(* Logix 5000 project; controller reports 1756-L63 rev 20.15; software revision 20.04; part 34 of 52 *)

        [22].log_data[35].max := 1.0, [22].log_data[35].total := 1322.998, [22].log_data[35].time := 3600.0, [22].log_data[35].minminute := 3, [22].log_data[35].valid := 1, [22].log_data[36].max := 1.0, [22].log_data[36].total := 1539.2471, [22].log_data[36].time := 3600.0, [22].log_data[36].maxminute := 5, [22].log_data[36].valid := 1, [22].log_data[37].time := 3600.0, [22].log_data[37].valid := 1, [22].log_data[38].time := 3600.0, [22].log_data[38].valid := 1, [22].log_data[39].min := 0.9938818, [22].log_data[39].max := 1.0064838, [22].log_data[39].total := 3605.8333, [22].log_data[39].time := 3600.0, [22].log_data[39].minminute := 45, [22].log_data[39].maxminute := 14, [22].log_data[39].valid := 1, [22].log_data[40].min := 7.5643167, [22].log_data[40].max := 7.586301, [22].log_data[40].total := 27282.406, [22].log_data[40].time := 3600.0, [22].log_data[40].minminute := 14, [22].log_data[40].maxminute := 26, [22].log_data[40].valid := 1, [22].log_data[41].min := 0.032943603, [22].log_data[41].max := 0.058854003, [22].log_data[41].total := 164.49648, [22].log_data[41].time := 3600.0, [22].log_data[41].minminute := 22, [22].log_data[41].valid := 1, [22].log_data[42].min := 2.291996, [22].log_data[42].max := 2.297767, [22].log_data[42].total := 8263.503, [22].log_data[42].time := 3600.0, [22].log_data[42].minminute := 32, [22].log_data[42].maxminute := 12, [22].log_data[42].valid := 1, [22].log_data[43].min := -0.26000214, [22].log_data[43].max := -0.26000214, [22].log_data[43].total := -935.9732, [22].log_data[43].time := 3600.0, [22].log_data[43].valid := 1, [22].log_data[44].min := -0.30000305, [22].log_data[44].max := -0.27999878, [22].log_data[44].total := -1015.7973, [22].log_data[44].time := 3600.0, [22].log_data[44].valid := 1, [22].log_data[45].time := 3600.0, [22].log_data[45].valid := 1, [22].log_data[46].time := 3600.0, [22].log_data[46].valid := 1, [22].log_data[47].time := 3600.0, [22].log_data[47].valid := 1, [22].log_data[48].min := 6.7563815, [22].log_data[48].max := 6.7984266, [22].log_data[48].total := 24360.947,
        [22].log_data[48].time := 3600.0, [22].log_data[48].minminute := 57, [22].log_data[48].valid := 1, [22].log_data[49].min := 8.905314, [22].log_data[49].max := 9.548168, [22].log_data[49].total := 33928.742, [22].log_data[49].time := 3600.0, [22].log_data[49].maxminute := 53, [22].log_data[49].valid := 1, [22].log_data[50].min := 1.9997966, [22].log_data[50].max := 2.0873032, [22].log_data[50].total := 7348.6255, [22].log_data[50].time := 3600.0, [22].log_data[50].minminute := 54, [22].log_data[50].maxminute := 59, [22].log_data[50].valid := 1, [22].log_data[51].time := 3600.0, [22].log_data[51].valid := 1, [22].log_data[52].min := -2.7799988, [22].log_data[52].max := 0.13999939, [22].log_data[52].total := -7224.4995, [22].log_data[52].time := 3600.0, [22].log_data[52].minminute := 27, [22].log_data[52].valid := 1, [22].log_data[53].min := -2.7000046, [22].log_data[53].max := 0.19999695, [22].log_data[53].total := -6896.3794, [22].log_data[53].time := 3600.0, [22].log_data[53].minminute := 16, [22].log_data[53].maxminute := 5, [22].log_data[53].valid := 1, [22].log_data[54].max := 0.537, [22].log_data[54].total := 1118.8905, [22].log_data[54].time := 3600.0, [22].log_data[54].valid := 1, [22].log_data[55].max := 0.5575, [22].log_data[55].total := 1135.9928, [22].log_data[55].time := 3600.0, [22].log_data[55].minminute := 3, [22].log_data[55].maxminute := 16, [22].log_data[55].valid := 1, [22].log_data[56].min := 0.16024561, [22].log_data[56].max := 0.1607167, [22].log_data[56].total := 577.52075, [22].log_data[56].time := 3600.0, [22].log_data[56].minminute := 12, [22].log_data[56].maxminute := 46, [22].log_data[56].valid := 1, [22].log_data[57].min := 0.3022821, [22].log_data[57].max := 0.30271393, [22].log_data[57].total := 1088.9108, [22].log_data[57].time := 3600.0, [22].log_data[57].minminute := 44, [22].log_data[57].maxminute := 4, [22].log_data[57].valid := 1, [22].log_data[58].time := 3600.0, [22].log_data[58].valid := 1, [22].log_data[59].time := 3600.0, [22].log_data[59].valid := 1, [22].log_data[60].valid := 1,
        [22].log_data[61].valid := 1, [22].log_data[62].valid := 1, [22].log_data[63].valid := 1, [22].log_data[64].valid := 1, [22].log_data[65].valid := 1, [22].log_data[66].valid := 1, [22].log_data[67].valid := 1, [22].log_data[68].valid := 1, [22].log_data[69].valid := 1, [22].log_data[70].valid := 1, [22].log_data[71].valid := 1, [22].log_data[72].valid := 1, [22].log_data[73].valid := 1, [22].log_data[74].valid := 1, [22].log_data[75].valid := 1, [22].log_data[76].valid := 1, [22].log_data[77].valid := 1, [22].log_data[78].valid := 1, [22].log_data[79].valid := 1, [22].log_data[80].valid := 1, [22].log_data[81].valid := 1, [22].log_data[82].valid := 1, [22].log_data[83].valid := 1, [22].log_data[84].valid := 1, [22].log_data[85].valid := 1, [22].log_data[86].valid := 1, [22].log_data[87].valid := 1, [22].log_data[88].valid := 1, [22].log_data[89].valid := 1, [22].log_data[90].valid := 1, [22].log_data[91].valid := 1, [22].log_data[92].valid := 1, [22].log_data[93].valid := 1, [22].log_data[94].valid := 1, [22].log_data[95].valid := 1, [22].log_data[96].valid := 1, [22].log_data[97].valid := 1, [22].log_data[98].valid := 1, [22].log_data[99].valid := 1, [22].log_data[100].valid := 1, [22].log_data[101].valid := 1, [22].log_data[102].valid := 1, [22].log_data[103].valid := 1, [22].log_data[104].valid := 1, [22].log_data[105].valid := 1, [22].log_data[106].valid := 1, [22].log_data[107].valid := 1, [22].log_data[108].valid := 1, [22].log_data[109].valid := 1, [22].log_data[110].valid := 1, [22].log_data[111].valid := 1, [22].log_data[112].valid := 1, [22].log_data[113].valid := 1, [22].log_data[114].valid := 1, [22].log_data[115].valid := 1, [22].log_data[116].valid := 1, [22].log_data[117].valid := 1, [22].log_data[118].valid := 1, [22].log_data[119].valid := 1, [22].log_data[120].valid := 1,
        [22].log_data[121].valid := 1, [22].log_data[122].valid := 1, [22].log_data[123].valid := 1, [22].log_data[124].valid := 1, [22].time.Year := 2023, [22].time.Month := 1, [22].time.Day := 14, [22].time.Hour := 1, [22].time.Minute := 59, [22].time.Second := 59, [23].log_data[0].min := 1.0, [23].log_data[0].max := 1.0, [23].log_data[0].total := 3600.0, [23].log_data[0].time := 3600.0, [23].log_data[0].valid := 1, [23].log_data[1].max := 1.0, [23].log_data[1].total := 523.5, [23].log_data[1].time := 3600.0, [23].log_data[1].maxminute := 36, [23].log_data[1].valid := 1, [23].log_data[2].max := 1.0, [23].log_data[2].total := 520.0, [23].log_data[2].time := 3600.0, [23].log_data[2].maxminute := 36, [23].log_data[2].valid := 1, [23].log_data[3].time := 3600.0, [23].log_data[3].valid := 1, [23].log_data[4].time := 3600.0, [23].log_data[4].valid := 1, [23].log_data[5].max := 1.0, [23].log_data[5].total := 229.5, [23].log_data[5].time := 3600.0, [23].log_data[5].maxminute := 39, [23].log_data[5].valid := 1, [23].log_data[6].time := 3600.0, [23].log_data[6].valid := 1, [23].log_data[7].time := 3600.0, [23].log_data[7].valid := 1, [23].log_data[8].max := 1.0, [23].log_data[8].total := 1148.249, [23].log_data[8].time := 3600.0, [23].log_data[8].maxminute := 40, [23].log_data[8].valid := 1, [23].log_data[9].max := 1.0, [23].log_data[9].total := 1144.749, [23].log_data[9].time := 3600.0, [23].log_data[9].maxminute := 40, [23].log_data[9].valid := 1, [23].log_data[10].min := 1.0, [23].log_data[10].max := 1.0, [23].log_data[10].total := 3600.0, [23].log_data[10].time := 3600.0, [23].log_data[10].valid := 1, [23].log_data[11].time := 3600.0, [23].log_data[11].valid := 1, [23].log_data[12].min := 1.0, [23].log_data[12].max := 1.0, [23].log_data[12].total := 3600.0, [23].log_data[12].time := 3600.0, [23].log_data[12].valid := 1,
        [23].log_data[13].min := 1.0, [23].log_data[13].max := 1.0, [23].log_data[13].total := 3600.0, [23].log_data[13].time := 3600.0, [23].log_data[13].valid := 1, [23].log_data[14].time := 3600.0, [23].log_data[14].valid := 1, [23].log_data[15].time := 3600.0, [23].log_data[15].valid := 1, [23].log_data[16].time := 3600.0, [23].log_data[16].valid := 1, [23].log_data[17].min := 1.0, [23].log_data[17].max := 1.0, [23].log_data[17].total := 3600.0, [23].log_data[17].time := 3600.0, [23].log_data[17].valid := 1, [23].log_data[18].time := 3600.0, [23].log_data[18].valid := 1, [23].log_data[19].time := 3600.0, [23].log_data[19].valid := 1, [23].log_data[20].time := 3600.0, [23].log_data[20].valid := 1, [23].log_data[21].min := 1.0, [23].log_data[21].max := 1.0, [23].log_data[21].total := 3600.0, [23].log_data[21].time := 3600.0, [23].log_data[21].valid := 1, [23].log_data[22].time := 3600.0, [23].log_data[22].valid := 1, [23].log_data[23].time := 3600.0, [23].log_data[23].valid := 1, [23].log_data[24].time := 3600.0, [23].log_data[24].valid := 1, [23].log_data[25].time := 3600.0, [23].log_data[25].valid := 1, [23].log_data[26].time := 3600.0, [23].log_data[26].valid := 1, [23].log_data[27].time := 3600.0, [23].log_data[27].valid := 1, [23].log_data[28].time := 3600.0, [23].log_data[28].valid := 1, [23].log_data[29].min := 1.0, [23].log_data[29].max := 1.0, [23].log_data[29].total := 3600.0, [23].log_data[29].time := 3600.0, [23].log_data[29].valid := 1, [23].log_data[30].min := 1.0, [23].log_data[30].max := 1.0, [23].log_data[30].total := 3600.0, [23].log_data[30].time := 3600.0, [23].log_data[30].valid := 1, [23].log_data[31].max := 1.0, [23].log_data[31].total := 434.5, [23].log_data[31].time := 3600.0, [23].log_data[31].maxminute := 40, [23].log_data[31].valid := 1, [23].log_data[32].max := 1.0, [23].log_data[32].total := 543.249, [23].log_data[32].time := 3600.0, [23].log_data[32].maxminute := 49,
        [23].log_data[32].valid := 1, [23].log_data[33].time := 3600.0, [23].log_data[33].valid := 1, [23].log_data[34].time := 3600.0, [23].log_data[34].valid := 1, [23].log_data[35].max := 1.0, [23].log_data[35].total := 417.998, [23].log_data[35].time := 3600.0, [23].log_data[35].maxminute := 41, [23].log_data[35].valid := 1, [23].log_data[36].max := 1.0, [23].log_data[36].total := 543.249, [23].log_data[36].time := 3600.0, [23].log_data[36].maxminute := 44, [23].log_data[36].valid := 1, [23].log_data[37].max := 7.614469, [23].log_data[37].total := 3441.945, [23].log_data[37].time := 3600.0, [23].log_data[37].maxminute := 38, [23].log_data[37].valid := 1, [23].log_data[38].time := 3600.0, [23].log_data[38].valid := 1, [23].log_data[39].min := 0.9950596, [23].log_data[39].max := 1.02203, [23].log_data[39].total := 3610.5056, [23].log_data[39].time := 3600.0, [23].log_data[39].minminute := 11, [23].log_data[39].maxminute := 43, [23].log_data[39].valid := 1, [23].log_data[40].min := 7.5431566, [23].log_data[40].max := 7.5961943, [23].log_data[40].total := 27280.893, [23].log_data[40].time := 3600.0, [23].log_data[40].minminute := 4, [23].log_data[40].maxminute := 36, [23].log_data[40].valid := 1, [23].log_data[41].min := 0.030784423, [23].log_data[41].max := 0.052769043, [23].log_data[41].total := 143.54086, [23].log_data[41].time := 3600.0, [23].log_data[41].minminute := 33, [23].log_data[41].maxminute := 9, [23].log_data[41].valid := 1, [23].log_data[42].min := 2.291996, [23].log_data[42].max := 2.2975314, [23].log_data[42].total := 8263.341, [23].log_data[42].time := 3600.0, [23].log_data[42].minminute := 5, [23].log_data[42].maxminute := 10, [23].log_data[42].valid := 1, [23].log_data[43].min := -0.26000214, [23].log_data[43].max := -0.26000214, [23].log_data[43].total := -935.9732, [23].log_data[43].time := 3600.0, [23].log_data[43].valid := 1, [23].log_data[44].min := -0.30000305, [23].log_data[44].max := -0.27999878, [23].log_data[44].total := -1011.4277, [23].log_data[44].time := 3600.0, [23].log_data[44].valid := 1,
        [23].log_data[45].time := 3600.0, [23].log_data[45].valid := 1, [23].log_data[46].time := 3600.0, [23].log_data[46].valid := 1, [23].log_data[47].time := 3600.0, [23].log_data[47].valid := 1, [23].log_data[48].min := 6.665145, [23].log_data[48].max := 6.9523196, [23].log_data[48].total := 24385.578, [23].log_data[48].time := 3600.0, [23].log_data[48].minminute := 59, [23].log_data[48].maxminute := 45, [23].log_data[48].valid := 1, [23].log_data[49].min := 7.0688124, [23].log_data[49].max := 9.542084, [23].log_data[49].total := 32485.41, [23].log_data[49].time := 3600.0, [23].log_data[49].minminute := 59, [23].log_data[49].maxminute := 3, [23].log_data[49].valid := 1, [23].log_data[50].min := 2.0678706, [23].log_data[50].max := 2.1526685, [23].log_data[50].total := 7561.778, [23].log_data[50].time := 3600.0, [23].log_data[50].minminute := 43, [23].log_data[50].maxminute := 40, [23].log_data[50].valid := 1, [23].log_data[51].time := 3600.0, [23].log_data[51].valid := 1, [23].log_data[52].min := -4.1800003, [23].log_data[52].max := 0.11999512, [23].log_data[52].total := -6155.475, [23].log_data[52].time := 3600.0, [23].log_data[52].minminute := 41, [23].log_data[52].maxminute := 48, [23].log_data[52].valid := 1, [23].log_data[53].min := -3.9799957, [23].log_data[53].max := 0.19999695, [23].log_data[53].total := -5728.4756, [23].log_data[53].time := 3600.0, [23].log_data[53].minminute := 41, [23].log_data[53].maxminute := 54, [23].log_data[53].valid := 1, [23].log_data[54].max := 0.5275, [23].log_data[54].total := 387.55862, [23].log_data[54].time := 3600.0, [23].log_data[54].maxminute := 49, [23].log_data[54].valid := 1, [23].log_data[55].max := 0.5285, [23].log_data[55].total := 378.56726, [23].log_data[55].time := 3600.0, [23].log_data[55].maxminute := 54, [23].log_data[55].valid := 1, [23].log_data[56].min := 0.16024561, [23].log_data[56].max := 0.1607167, [23].log_data[56].total := 577.70746, [23].log_data[56].time := 3600.0, [23].log_data[56].minminute := 54, [23].log_data[56].maxminute := 30, [23].log_data[56].valid := 1,
        [23].log_data[57].min := 0.30232134, [23].log_data[57].max := 0.30275318, [23].log_data[57].total := 1088.9501, [23].log_data[57].time := 3600.0, [23].log_data[57].maxminute := 43, [23].log_data[57].valid := 1, [23].log_data[58].time := 3600.0, [23].log_data[58].valid := 1, [23].log_data[59].time := 3600.0, [23].log_data[59].valid := 1, [23].log_data[60].valid := 1, [23].log_data[61].valid := 1, [23].log_data[62].valid := 1, [23].log_data[63].valid := 1, [23].log_data[64].valid := 1, [23].log_data[65].valid := 1, [23].log_data[66].valid := 1, [23].log_data[67].valid := 1, [23].log_data[68].valid := 1, [23].log_data[69].valid := 1, [23].log_data[70].valid := 1, [23].log_data[71].valid := 1, [23].log_data[72].valid := 1, [23].log_data[73].valid := 1, [23].log_data[74].valid := 1, [23].log_data[75].valid := 1, [23].log_data[76].valid := 1, [23].log_data[77].valid := 1, [23].log_data[78].valid := 1, [23].log_data[79].valid := 1, [23].log_data[80].valid := 1, [23].log_data[81].valid := 1, [23].log_data[82].valid := 1, [23].log_data[83].valid := 1, [23].log_data[84].valid := 1, [23].log_data[85].valid := 1, [23].log_data[86].valid := 1, [23].log_data[87].valid := 1, [23].log_data[88].valid := 1, [23].log_data[89].valid := 1, [23].log_data[90].valid := 1, [23].log_data[91].valid := 1, [23].log_data[92].valid := 1, [23].log_data[93].valid := 1, [23].log_data[94].valid := 1, [23].log_data[95].valid := 1, [23].log_data[96].valid := 1, [23].log_data[97].valid := 1, [23].log_data[98].valid := 1, [23].log_data[99].valid := 1, [23].log_data[100].valid := 1, [23].log_data[101].valid := 1, [23].log_data[102].valid := 1, [23].log_data[103].valid := 1, [23].log_data[104].valid := 1, [23].log_data[105].valid := 1, [23].log_data[106].valid := 1, [23].log_data[107].valid := 1, [23].log_data[108].valid := 1, [23].log_data[109].valid := 1,
        [23].log_data[110].valid := 1, [23].log_data[111].valid := 1, [23].log_data[112].valid := 1, [23].log_data[113].valid := 1, [23].log_data[114].valid := 1, [23].log_data[115].valid := 1, [23].log_data[116].valid := 1, [23].log_data[117].valid := 1, [23].log_data[118].valid := 1, [23].log_data[119].valid := 1, [23].log_data[120].valid := 1, [23].log_data[121].valid := 1, [23].log_data[122].valid := 1, [23].log_data[123].valid := 1, [23].log_data[124].valid := 1, [23].time.Year := 2023, [23].time.Month := 1, [23].time.Day := 14, [23].time.Hour := 2, [23].time.Minute := 59, [23].time.Second := 59, [24].log_data[0].min := 1.0, [24].log_data[0].max := 1.0, [24].log_data[0].total := 3600.0, [24].log_data[0].time := 3600.0, [24].log_data[0].valid := 1, [24].log_data[1].time := 3600.0, [24].log_data[1].valid := 1, [24].log_data[2].time := 3600.0, [24].log_data[2].valid := 1, [24].log_data[3].time := 3600.0, [24].log_data[3].valid := 1, [24].log_data[4].time := 3600.0, [24].log_data[4].valid := 1, [24].log_data[5].time := 3600.0, [24].log_data[5].valid := 1, [24].log_data[6].time := 3600.0, [24].log_data[6].valid := 1, [24].log_data[7].time := 3600.0, [24].log_data[7].valid := 1, [24].log_data[8].min := 1.0, [24].log_data[8].max := 1.0, [24].log_data[8].total := 3600.0, [24].log_data[8].time := 3600.0, [24].log_data[8].valid := 1, [24].log_data[9].min := 1.0, [24].log_data[9].max := 1.0, [24].log_data[9].total := 3600.0, [24].log_data[9].time := 3600.0, [24].log_data[9].valid := 1, [24].log_data[10].min := 1.0, [24].log_data[10].max := 1.0, [24].log_data[10].total := 3600.0, [24].log_data[10].time := 3600.0, [24].log_data[10].valid := 1, [24].log_data[11].time := 3600.0, [24].log_data[11].valid := 1, [24].log_data[12].min := 1.0, [24].log_data[12].max := 1.0, [24].log_data[12].total := 3600.0,
        [24].log_data[12].time := 3600.0, [24].log_data[12].valid := 1, [24].log_data[13].min := 1.0, [24].log_data[13].max := 1.0, [24].log_data[13].total := 3600.0, [24].log_data[13].time := 3600.0, [24].log_data[13].valid := 1, [24].log_data[14].time := 3600.0, [24].log_data[14].valid := 1, [24].log_data[15].time := 3600.0, [24].log_data[15].valid := 1, [24].log_data[16].time := 3600.0, [24].log_data[16].valid := 1, [24].log_data[17].min := 1.0, [24].log_data[17].max := 1.0, [24].log_data[17].total := 3600.0, [24].log_data[17].time := 3600.0, [24].log_data[17].valid := 1, [24].log_data[18].time := 3600.0, [24].log_data[18].valid := 1, [24].log_data[19].time := 3600.0, [24].log_data[19].valid := 1, [24].log_data[20].time := 3600.0, [24].log_data[20].valid := 1, [24].log_data[21].min := 1.0, [24].log_data[21].max := 1.0, [24].log_data[21].total := 3600.0, [24].log_data[21].time := 3600.0, [24].log_data[21].valid := 1, [24].log_data[22].time := 3600.0, [24].log_data[22].valid := 1, [24].log_data[23].time := 3600.0, [24].log_data[23].valid := 1, [24].log_data[24].time := 3600.0, [24].log_data[24].valid := 1, [24].log_data[25].time := 3600.0, [24].log_data[25].valid := 1, [24].log_data[26].time := 3600.0, [24].log_data[26].valid := 1, [24].log_data[27].time := 3600.0, [24].log_data[27].valid := 1, [24].log_data[28].time := 3600.0, [24].log_data[28].valid := 1, [24].log_data[29].min := 1.0, [24].log_data[29].max := 1.0, [24].log_data[29].total := 3600.0, [24].log_data[29].time := 3600.0, [24].log_data[29].valid := 1, [24].log_data[30].min := 1.0, [24].log_data[30].max := 1.0, [24].log_data[30].total := 3600.0, [24].log_data[30].time := 3600.0, [24].log_data[30].valid := 1, [24].log_data[31].max := 1.0, [24].log_data[31].total := 1629.7471, [24].log_data[31].time := 3600.0, [24].log_data[31].valid := 1, [24].log_data[32].max := 1.0, [24].log_data[32].total := 1515.7471, [24].log_data[32].time := 3600.0,
        [24].log_data[32].maxminute := 10, [24].log_data[32].valid := 1, [24].log_data[33].time := 3600.0, [24].log_data[33].valid := 1, [24].log_data[34].time := 3600.0, [24].log_data[34].valid := 1, [24].log_data[35].max := 1.0, [24].log_data[35].total := 1440.7471, [24].log_data[35].time := 3600.0, [24].log_data[35].minminute := 3, [24].log_data[35].valid := 1, [24].log_data[36].max := 1.0, [24].log_data[36].total := 1629.7471, [24].log_data[36].time := 3600.0, [24].log_data[36].maxminute := 5, [24].log_data[36].valid := 1, [24].log_data[37].time := 3600.0, [24].log_data[37].valid := 1, [24].log_data[38].time := 3600.0, [24].log_data[38].valid := 1, [24].log_data[39].min := 0.9945885, [24].log_data[39].max := 1.0074259, [24].log_data[39].total := 3607.058, [24].log_data[39].time := 3600.0, [24].log_data[39].minminute := 14, [24].log_data[39].maxminute := 34, [24].log_data[39].valid := 1, [24].log_data[40].min := 7.5717363, [24].log_data[40].max := 7.586301, [24].log_data[40].total := 27285.361, [24].log_data[40].time := 3600.0, [24].log_data[40].minminute := 3, [24].log_data[40].maxminute := 5, [24].log_data[40].valid := 1, [24].log_data[41].min := 0.029017823, [24].log_data[41].max := 0.047469236, [24].log_data[41].total := 144.30215, [24].log_data[41].time := 3600.0, [24].log_data[41].minminute := 46, [24].log_data[41].maxminute := 11, [24].log_data[41].valid := 1, [24].log_data[42].min := 2.292585, [24].log_data[42].max := 2.297767, [24].log_data[42].total := 8263.188, [24].log_data[42].time := 3600.0, [24].log_data[42].minminute := 8, [24].log_data[42].maxminute := 13, [24].log_data[42].valid := 1, [24].log_data[43].min := -0.26000214, [24].log_data[43].max := -0.26000214, [24].log_data[43].total := -935.9732, [24].log_data[43].time := 3600.0, [24].log_data[43].valid := 1, [24].log_data[44].min := -0.30000305, [24].log_data[44].max := -0.27999878, [24].log_data[44].total := -1011.2831, [24].log_data[44].time := 3600.0, [24].log_data[44].valid := 1, [24].log_data[45].time := 3600.0, [24].log_data[45].valid := 1,
        [24].log_data[46].time := 3600.0, [24].log_data[46].valid := 1, [24].log_data[47].time := 3600.0, [24].log_data[47].valid := 1, [24].log_data[48].min := 6.595069, [24].log_data[48].max := 6.7967777, [24].log_data[48].total := 24212.92, [24].log_data[48].time := 3600.0, [24].log_data[48].minminute := 10, [24].log_data[48].maxminute := 25, [24].log_data[48].valid := 1, [24].log_data[49].min := 6.9688993, [24].log_data[49].max := 9.5318775, [24].log_data[49].total := 31036.44, [24].log_data[49].time := 3600.0, [24].log_data[49].minminute := 2, [24].log_data[49].maxminute := 58, [24].log_data[49].valid := 1, [24].log_data[50].min := 2.006863, [24].log_data[50].max := 2.0901299, [24].log_data[50].total := 7375.6206, [24].log_data[50].time := 3600.0, [24].log_data[50].minminute := 59, [24].log_data[50].valid := 1, [24].log_data[51].time := 3600.0, [24].log_data[51].valid := 1, [24].log_data[52].min := -3.040001, [24].log_data[52].max := 0.13999939, [24].log_data[52].total := -7732.567, [24].log_data[52].time := 3600.0, [24].log_data[52].minminute := 42, [24].log_data[52].maxminute := 40, [24].log_data[52].valid := 1, [24].log_data[53].min := -2.5, [24].log_data[53].max := 0.22000122, [24].log_data[53].total := -7008.48, [24].log_data[53].time := 3600.0, [24].log_data[53].minminute := 18, [24].log_data[53].maxminute := 4, [24].log_data[53].valid := 1, [24].log_data[54].max := 0.5645, [24].log_data[54].total := 1246.528, [24].log_data[54].time := 3600.0, [24].log_data[54].maxminute := 42, [24].log_data[54].valid := 1, [24].log_data[55].max := 0.538, [24].log_data[55].total := 1217.1504, [24].log_data[55].time := 3600.0, [24].log_data[55].minminute := 3, [24].log_data[55].maxminute := 47, [24].log_data[55].valid := 1, [24].log_data[56].min := 0.16024561, [24].log_data[56].max := 0.16079521, [24].log_data[56].total := 577.71893, [24].log_data[56].time := 3600.0, [24].log_data[56].minminute := 56, [24].log_data[56].maxminute := 32, [24].log_data[56].valid := 1, [24].log_data[57].min := 0.30079022, [24].log_data[57].max := 0.30271393,
        [24].log_data[57].total := 1084.8229, [24].log_data[57].time := 3600.0, [24].log_data[57].minminute := 47, [24].log_data[57].valid := 1, [24].log_data[58].time := 3600.0, [24].log_data[58].valid := 1, [24].log_data[59].time := 3600.0, [24].log_data[59].valid := 1, [24].log_data[60].valid := 1, [24].log_data[61].valid := 1, [24].log_data[62].valid := 1, [24].log_data[63].valid := 1, [24].log_data[64].valid := 1, [24].log_data[65].valid := 1, [24].log_data[66].valid := 1, [24].log_data[67].valid := 1, [24].log_data[68].valid := 1, [24].log_data[69].valid := 1, [24].log_data[70].valid := 1, [24].log_data[71].valid := 1, [24].log_data[72].valid := 1, [24].log_data[73].valid := 1, [24].log_data[74].valid := 1, [24].log_data[75].valid := 1, [24].log_data[76].valid := 1, [24].log_data[77].valid := 1, [24].log_data[78].valid := 1, [24].log_data[79].valid := 1, [24].log_data[80].valid := 1, [24].log_data[81].valid := 1, [24].log_data[82].valid := 1, [24].log_data[83].valid := 1, [24].log_data[84].valid := 1, [24].log_data[85].valid := 1, [24].log_data[86].valid := 1, [24].log_data[87].valid := 1, [24].log_data[88].valid := 1, [24].log_data[89].valid := 1, [24].log_data[90].valid := 1, [24].log_data[91].valid := 1, [24].log_data[92].valid := 1, [24].log_data[93].valid := 1, [24].log_data[94].valid := 1, [24].log_data[95].valid := 1, [24].log_data[96].valid := 1, [24].log_data[97].valid := 1, [24].log_data[98].valid := 1, [24].log_data[99].valid := 1, [24].log_data[100].valid := 1, [24].log_data[101].valid := 1, [24].log_data[102].valid := 1, [24].log_data[103].valid := 1, [24].log_data[104].valid := 1, [24].log_data[105].valid := 1, [24].log_data[106].valid := 1, [24].log_data[107].valid := 1, [24].log_data[108].valid := 1, [24].log_data[109].valid := 1, [24].log_data[110].valid := 1, [24].log_data[111].valid := 1,
        [24].log_data[112].valid := 1, [24].log_data[113].valid := 1, [24].log_data[114].valid := 1, [24].log_data[115].valid := 1, [24].log_data[116].valid := 1, [24].log_data[117].valid := 1, [24].log_data[118].valid := 1, [24].log_data[119].valid := 1, [24].log_data[120].valid := 1, [24].log_data[121].valid := 1, [24].log_data[122].valid := 1, [24].log_data[123].valid := 1, [24].log_data[124].valid := 1, [24].time.Year := 2023, [24].time.Month := 1, [24].time.Day := 14, [24].time.Hour := 3, [24].time.Minute := 59, [24].time.Second := 59, [25].log_data[0].min := 1.0, [25].log_data[0].max := 1.0, [25].log_data[0].total := 3600.0, [25].log_data[0].time := 3600.0, [25].log_data[0].valid := 1, [25].log_data[1].time := 3600.0, [25].log_data[1].valid := 1, [25].log_data[2].time := 3600.0, [25].log_data[2].valid := 1, [25].log_data[3].time := 3600.0, [25].log_data[3].valid := 1, [25].log_data[4].time := 3600.0, [25].log_data[4].valid := 1, [25].log_data[5].time := 3600.0, [25].log_data[5].valid := 1, [25].log_data[6].time := 3600.0, [25].log_data[6].valid := 1, [25].log_data[7].time := 3600.0, [25].log_data[7].valid := 1, [25].log_data[8].max := 1.0, [25].log_data[8].total := 227.751, [25].log_data[8].time := 3600.0, [25].log_data[8].minminute := 3, [25].log_data[8].valid := 1, [25].log_data[9].max := 1.0, [25].log_data[9].total := 227.751, [25].log_data[9].time := 3600.0, [25].log_data[9].minminute := 3, [25].log_data[9].valid := 1, [25].log_data[10].min := 1.0, [25].log_data[10].max := 1.0, [25].log_data[10].total := 3600.0, [25].log_data[10].time := 3600.0, [25].log_data[10].valid := 1, [25].log_data[11].time := 3600.0, [25].log_data[11].valid := 1, [25].log_data[12].min := 1.0, [25].log_data[12].max := 1.0, [25].log_data[12].total := 3600.0, [25].log_data[12].time := 3600.0, [25].log_data[12].valid := 1,
        [25].log_data[13].min := 1.0, [25].log_data[13].max := 1.0, [25].log_data[13].total := 3600.0, [25].log_data[13].time := 3600.0, [25].log_data[13].valid := 1, [25].log_data[14].time := 3600.0, [25].log_data[14].valid := 1, [25].log_data[15].time := 3600.0, [25].log_data[15].valid := 1, [25].log_data[16].time := 3600.0, [25].log_data[16].valid := 1, [25].log_data[17].min := 1.0, [25].log_data[17].max := 1.0, [25].log_data[17].total := 3600.0, [25].log_data[17].time := 3600.0, [25].log_data[17].valid := 1, [25].log_data[18].time := 3600.0, [25].log_data[18].valid := 1, [25].log_data[19].time := 3600.0, [25].log_data[19].valid := 1, [25].log_data[20].time := 3600.0, [25].log_data[20].valid := 1, [25].log_data[21].min := 1.0, [25].log_data[21].max := 1.0, [25].log_data[21].total := 3600.0, [25].log_data[21].time := 3600.0, [25].log_data[21].valid := 1, [25].log_data[22].time := 3600.0, [25].log_data[22].valid := 1, [25].log_data[23].time := 3600.0, [25].log_data[23].valid := 1, [25].log_data[24].time := 3600.0, [25].log_data[24].valid := 1, [25].log_data[25].time := 3600.0, [25].log_data[25].valid := 1, [25].log_data[26].time := 3600.0, [25].log_data[26].valid := 1, [25].log_data[27].time := 3600.0, [25].log_data[27].valid := 1, [25].log_data[28].time := 3600.0, [25].log_data[28].valid := 1, [25].log_data[29].min := 1.0, [25].log_data[29].max := 1.0, [25].log_data[29].total := 3600.0, [25].log_data[29].time := 3600.0, [25].log_data[29].valid := 1, [25].log_data[30].min := 1.0, [25].log_data[30].max := 1.0, [25].log_data[30].total := 3600.0, [25].log_data[30].time := 3600.0, [25].log_data[30].valid := 1, [25].log_data[31].max := 1.0, [25].log_data[31].total := 29.249, [25].log_data[31].time := 3600.0, [25].log_data[31].maxminute := 3, [25].log_data[31].valid := 1, [25].log_data[32].max := 1.0, [25].log_data[32].total := 114.0, [25].log_data[32].time := 3600.0, [25].log_data[32].minminute := 1,
        [25].log_data[32].valid := 1, [25].log_data[33].time := 3600.0, [25].log_data[33].valid := 1, [25].log_data[34].time := 3600.0, [25].log_data[34].valid := 1, [25].log_data[35].max := 1.0, [25].log_data[35].total := 231.5, [25].log_data[35].time := 3600.0, [25].log_data[35].minminute := 3, [25].log_data[35].valid := 1, [25].log_data[36].time := 3600.0, [25].log_data[36].valid := 1, [25].log_data[37].time := 3600.0, [25].log_data[37].valid := 1, [25].log_data[38].time := 3600.0, [25].log_data[38].valid := 1, [25].log_data[39].min := 0.9945885, [25].log_data[39].max := 1.0076615, [25].log_data[39].total := 3606.9658, [25].log_data[39].time := 3600.0, [25].log_data[39].minminute := 56, [25].log_data[39].maxminute := 27, [25].log_data[39].valid := 1, [25].log_data[40].min := 7.5643167, [25].log_data[40].max := 7.587675, [25].log_data[40].total := 27287.488, [25].log_data[40].time := 3600.0, [25].log_data[40].minminute := 47, [25].log_data[40].maxminute := 27, [25].log_data[40].valid := 1, [25].log_data[41].min := 0.034906495, [25].log_data[41].max := 0.05963916, [25].log_data[41].total := 160.86324, [25].log_data[41].time := 3600.0, [25].log_data[41].maxminute := 49, [25].log_data[41].valid := 1, [25].log_data[42].min := 2.2922316, [25].log_data[42].max := 2.2974136, [25].log_data[42].total := 8263.044, [25].log_data[42].time := 3600.0, [25].log_data[42].minminute := 25, [25].log_data[42].maxminute := 36, [25].log_data[42].valid := 1, [25].log_data[43].min := -0.26000214, [25].log_data[43].max := -0.26000214, [25].log_data[43].total := -935.9732, [25].log_data[43].time := 3600.0, [25].log_data[43].valid := 1, [25].log_data[44].min := -0.30000305, [25].log_data[44].max := -0.27999878, [25].log_data[44].total := -1009.182, [25].log_data[44].time := 3600.0, [25].log_data[44].valid := 1, [25].log_data[45].time := 3600.0, [25].log_data[45].valid := 1, [25].log_data[46].time := 3600.0, [25].log_data[46].valid := 1, [25].log_data[47].time := 3600.0, [25].log_data[47].valid := 1, [25].log_data[48].min := 6.7492356,
        [25].log_data[48].max := 6.762702, [25].log_data[48].total := 24321.047, [25].log_data[48].time := 3600.0, [25].log_data[48].minminute := 5, [25].log_data[48].maxminute := 52, [25].log_data[48].valid := 1, [25].log_data[49].min := 9.508125, [25].log_data[49].max := 9.581735, [25].log_data[49].total := 34331.49, [25].log_data[49].time := 3600.0, [25].log_data[49].minminute := 7, [25].log_data[49].maxminute := 57, [25].log_data[49].valid := 1, [25].log_data[50].min := 1.9999144, [25].log_data[50].max := 2.1099162, [25].log_data[50].total := 7540.0083, [25].log_data[50].time := 3600.0, [25].log_data[50].minminute := 3, [25].log_data[50].maxminute := 54, [25].log_data[50].valid := 1, [25].log_data[51].time := 3600.0, [25].log_data[51].valid := 1, [25].log_data[52].min := -2.7400055, [25].log_data[52].max := 0.11999512, [25].log_data[52].total := -5230.148, [25].log_data[52].time := 3600.0, [25].log_data[52].minminute := 3, [25].log_data[52].maxminute := 2, [25].log_data[52].valid := 1, [25].log_data[53].min := -2.4800034, [25].log_data[53].max := -0.16000366, [25].log_data[53].total := -5175.728, [25].log_data[53].time := 3600.0, [25].log_data[53].maxminute := 3, [25].log_data[53].valid := 1, [25].log_data[54].max := 0.505, [25].log_data[54].total := 55.965687, [25].log_data[54].time := 3600.0, [25].log_data[54].minminute := 1, [25].log_data[54].maxminute := 3, [25].log_data[54].valid := 1, [25].log_data[55].max := 0.44349998, [25].log_data[55].total := 93.022255, [25].log_data[55].time := 3600.0, [25].log_data[55].minminute := 3, [25].log_data[55].valid := 1, [25].log_data[56].min := 0.16028486, [25].log_data[56].max := 0.16079521, [25].log_data[56].total := 577.82935, [25].log_data[56].time := 3600.0, [25].log_data[56].minminute := 2, [25].log_data[56].maxminute := 7, [25].log_data[56].valid := 1, [25].log_data[57].min := 0.3008295, [25].log_data[57].max := 0.30126134, [25].log_data[57].total := 1083.6661, [25].log_data[57].time := 3600.0, [25].log_data[57].minminute := 3, [25].log_data[57].maxminute := 28, [25].log_data[57].valid := 1,
        [25].log_data[58].time := 3600.0, [25].log_data[58].valid := 1, [25].log_data[59].time := 3600.0, [25].log_data[59].valid := 1, [25].log_data[60].valid := 1, [25].log_data[61].valid := 1, [25].log_data[62].valid := 1, [25].log_data[63].valid := 1, [25].log_data[64].valid := 1, [25].log_data[65].valid := 1, [25].log_data[66].valid := 1, [25].log_data[67].valid := 1, [25].log_data[68].valid := 1, [25].log_data[69].valid := 1, [25].log_data[70].valid := 1, [25].log_data[71].valid := 1, [25].log_data[72].valid := 1, [25].log_data[73].valid := 1, [25].log_data[74].valid := 1, [25].log_data[75].valid := 1, [25].log_data[76].valid := 1, [25].log_data[77].valid := 1, [25].log_data[78].valid := 1, [25].log_data[79].valid := 1, [25].log_data[80].valid := 1, [25].log_data[81].valid := 1, [25].log_data[82].valid := 1, [25].log_data[83].valid := 1, [25].log_data[84].valid := 1, [25].log_data[85].valid := 1, [25].log_data[86].valid := 1, [25].log_data[87].valid := 1, [25].log_data[88].valid := 1, [25].log_data[89].valid := 1, [25].log_data[90].valid := 1, [25].log_data[91].valid := 1, [25].log_data[92].valid := 1, [25].log_data[93].valid := 1, [25].log_data[94].valid := 1, [25].log_data[95].valid := 1, [25].log_data[96].valid := 1, [25].log_data[97].valid := 1, [25].log_data[98].valid := 1, [25].log_data[99].valid := 1, [25].log_data[100].valid := 1, [25].log_data[101].valid := 1, [25].log_data[102].valid := 1, [25].log_data[103].valid := 1, [25].log_data[104].valid := 1, [25].log_data[105].valid := 1, [25].log_data[106].valid := 1, [25].log_data[107].valid := 1, [25].log_data[108].valid := 1, [25].log_data[109].valid := 1, [25].log_data[110].valid := 1, [25].log_data[111].valid := 1, [25].log_data[112].valid := 1, [25].log_data[113].valid := 1, [25].log_data[114].valid := 1, [25].log_data[115].valid := 1,
        [25].log_data[116].valid := 1, [25].log_data[117].valid := 1, [25].log_data[118].valid := 1, [25].log_data[119].valid := 1, [25].log_data[120].valid := 1, [25].log_data[121].valid := 1, [25].log_data[122].valid := 1, [25].log_data[123].valid := 1, [25].log_data[124].valid := 1, [25].time.Year := 2023, [25].time.Month := 1, [25].time.Day := 14, [25].time.Hour := 4, [25].time.Minute := 59, [25].time.Second := 59, [26].log_data[0].min := 1.0, [26].log_data[0].max := 1.0, [26].log_data[0].total := 3600.0, [26].log_data[0].time := 3600.0, [26].log_data[0].valid := 1, [26].log_data[1].time := 3600.0, [26].log_data[1].valid := 1, [26].log_data[2].time := 3600.0, [26].log_data[2].valid := 1, [26].log_data[3].time := 3600.0, [26].log_data[3].valid := 1, [26].log_data[4].time := 3600.0, [26].log_data[4].valid := 1, [26].log_data[5].time := 3600.0, [26].log_data[5].valid := 1, [26].log_data[6].time := 3600.0, [26].log_data[6].valid := 1, [26].log_data[7].time := 3600.0, [26].log_data[7].valid := 1, [26].log_data[8].time := 3600.0, [26].log_data[8].valid := 1, [26].log_data[9].time := 3600.0, [26].log_data[9].valid := 1, [26].log_data[10].min := 1.0, [26].log_data[10].max := 1.0, [26].log_data[10].total := 3600.0, [26].log_data[10].time := 3600.0, [26].log_data[10].valid := 1, [26].log_data[11].time := 3600.0, [26].log_data[11].valid := 1, [26].log_data[12].min := 1.0, [26].log_data[12].max := 1.0, [26].log_data[12].total := 3600.0, [26].log_data[12].time := 3600.0, [26].log_data[12].valid := 1, [26].log_data[13].min := 1.0, [26].log_data[13].max := 1.0, [26].log_data[13].total := 3600.0, [26].log_data[13].time := 3600.0, [26].log_data[13].valid := 1, [26].log_data[14].time := 3600.0, [26].log_data[14].valid := 1, [26].log_data[15].time := 3600.0, [26].log_data[15].valid := 1, [26].log_data[16].time := 3600.0,
        [26].log_data[16].valid := 1, [26].log_data[17].min := 1.0, [26].log_data[17].max := 1.0, [26].log_data[17].total := 3600.0, [26].log_data[17].time := 3600.0, [26].log_data[17].valid := 1, [26].log_data[18].time := 3600.0, [26].log_data[18].valid := 1, [26].log_data[19].time := 3600.0, [26].log_data[19].valid := 1, [26].log_data[20].time := 3600.0, [26].log_data[20].valid := 1, [26].log_data[21].min := 1.0, [26].log_data[21].max := 1.0, [26].log_data[21].total := 3600.0, [26].log_data[21].time := 3600.0, [26].log_data[21].valid := 1, [26].log_data[22].time := 3600.0, [26].log_data[22].valid := 1, [26].log_data[23].time := 3600.0, [26].log_data[23].valid := 1, [26].log_data[24].time := 3600.0, [26].log_data[24].valid := 1, [26].log_data[25].time := 3600.0, [26].log_data[25].valid := 1, [26].log_data[26].time := 3600.0, [26].log_data[26].valid := 1, [26].log_data[27].time := 3600.0, [26].log_data[27].valid := 1, [26].log_data[28].time := 3600.0, [26].log_data[28].valid := 1, [26].log_data[29].min := 1.0, [26].log_data[29].max := 1.0, [26].log_data[29].total := 3600.0, [26].log_data[29].time := 3600.0, [26].log_data[29].valid := 1, [26].log_data[30].min := 1.0, [26].log_data[30].max := 1.0, [26].log_data[30].total := 3600.0, [26].log_data[30].time := 3600.0, [26].log_data[30].valid := 1, [26].log_data[31].time := 3600.0, [26].log_data[31].valid := 1, [26].log_data[32].time := 3600.0, [26].log_data[32].valid := 1, [26].log_data[33].time := 3600.0, [26].log_data[33].valid := 1, [26].log_data[34].time := 3600.0, [26].log_data[34].valid := 1, [26].log_data[35].time := 3600.0, [26].log_data[35].valid := 1, [26].log_data[36].time := 3600.0, [26].log_data[36].valid := 1, [26].log_data[37].time := 3600.0, [26].log_data[37].valid := 1, [26].log_data[38].time := 3600.0, [26].log_data[38].valid := 1, [26].log_data[39].min := 0.99494183, [26].log_data[39].max := 1.0075438, [26].log_data[39].total := 3605.6262,
        [26].log_data[39].time := 3600.0, [26].log_data[39].minminute := 38, [26].log_data[39].maxminute := 35, [26].log_data[39].valid := 1, [26].log_data[40].min := 7.557446, [26].log_data[40].max := 7.597843, [26].log_data[40].total := 27287.11, [26].log_data[40].time := 3600.0, [26].log_data[40].minminute := 22, [26].log_data[40].maxminute := 25, [26].log_data[40].valid := 1, [26].log_data[41].min := 0.042954348, [26].log_data[41].max := 0.07396851, [26].log_data[41].total := 213.51753, [26].log_data[41].time := 3600.0, [26].log_data[41].minminute := 2, [26].log_data[41].maxminute := 53, [26].log_data[41].valid := 1, [26].log_data[42].min := 2.292467, [26].log_data[42].max := 2.2974136, [26].log_data[42].total := 8262.912, [26].log_data[42].time := 3600.0, [26].log_data[42].minminute := 16, [26].log_data[42].maxminute := 30, [26].log_data[42].valid := 1, [26].log_data[43].min := -0.26000214, [26].log_data[43].max := -0.23999786, [26].log_data[43].total := -935.9682, [26].log_data[43].time := 3600.0, [26].log_data[43].maxminute := 38, [26].log_data[43].valid := 1, [26].log_data[44].min := -0.30000305, [26].log_data[44].max := -0.27999878, [26].log_data[44].total := -1012.39764, [26].log_data[44].time := 3600.0, [26].log_data[44].valid := 1, [26].log_data[45].time := 3600.0, [26].log_data[45].valid := 1, [26].log_data[46].time := 3600.0, [26].log_data[46].valid := 1, [26].log_data[47].time := 3600.0, [26].log_data[47].valid := 1, [26].log_data[48].min := 6.7607784, [26].log_data[48].max := 6.774244, [26].log_data[48].total := 24362.328, [26].log_data[48].time := 3600.0, [26].log_data[48].maxminute := 54, [26].log_data[48].valid := 1, [26].log_data[49].min := 9.545813, [26].log_data[49].max := 9.615496, [26].log_data[49].total := 34480.9, [26].log_data[49].time := 3600.0, [26].log_data[49].minminute := 1, [26].log_data[49].maxminute := 58, [26].log_data[49].valid := 1, [26].log_data[50].min := 2.1028495, [26].log_data[50].max := 2.1112115, [26].log_data[50].total := 7590.1895, [26].log_data[50].time := 3600.0, [26].log_data[50].minminute := 24,
        [26].log_data[50].maxminute := 34, [26].log_data[50].valid := 1, [26].log_data[51].time := 3600.0, [26].log_data[51].valid := 1, [26].log_data[52].min := -1.5999985, [26].log_data[52].max := -1.4400024, [26].log_data[52].total := -5582.0986, [26].log_data[52].time := 3600.0, [26].log_data[52].minminute := 13, [26].log_data[52].maxminute := 3, [26].log_data[52].valid := 1, [26].log_data[53].min := -1.5600052, [26].log_data[53].max := -1.4000015, [26].log_data[53].total := -5329.579, [26].log_data[53].time := 3600.0, [26].log_data[53].minminute := 53, [26].log_data[53].valid := 1, [26].log_data[54].time := 3600.0, [26].log_data[54].valid := 1, [26].log_data[55].time := 3600.0, [26].log_data[55].valid := 1, [26].log_data[56].min := 0.16032413, [26].log_data[56].max := 0.16075596, [26].log_data[56].total := 577.7898, [26].log_data[56].time := 3600.0, [26].log_data[56].minminute := 31, [26].log_data[56].maxminute := 20, [26].log_data[56].valid := 1, [26].log_data[57].min := 0.300908, [26].log_data[57].max := 0.3013006, [26].log_data[57].total := 1083.8445, [26].log_data[57].time := 3600.0, [26].log_data[57].minminute := 1, [26].log_data[57].maxminute := 1, [26].log_data[57].valid := 1, [26].log_data[58].time := 3600.0, [26].log_data[58].valid := 1, [26].log_data[59].time := 3600.0, [26].log_data[59].valid := 1, [26].log_data[60].valid := 1, [26].log_data[61].valid := 1, [26].log_data[62].valid := 1, [26].log_data[63].valid := 1, [26].log_data[64].valid := 1, [26].log_data[65].valid := 1, [26].log_data[66].valid := 1, [26].log_data[67].valid := 1, [26].log_data[68].valid := 1, [26].log_data[69].valid := 1, [26].log_data[70].valid := 1, [26].log_data[71].valid := 1, [26].log_data[72].valid := 1, [26].log_data[73].valid := 1, [26].log_data[74].valid := 1, [26].log_data[75].valid := 1, [26].log_data[76].valid := 1, [26].log_data[77].valid := 1, [26].log_data[78].valid := 1, [26].log_data[79].valid := 1, [26].log_data[80].valid := 1,
        [26].log_data[81].valid := 1, [26].log_data[82].valid := 1, [26].log_data[83].valid := 1, [26].log_data[84].valid := 1, [26].log_data[85].valid := 1, [26].log_data[86].valid := 1, [26].log_data[87].valid := 1, [26].log_data[88].valid := 1, [26].log_data[89].valid := 1, [26].log_data[90].valid := 1, [26].log_data[91].valid := 1, [26].log_data[92].valid := 1, [26].log_data[93].valid := 1, [26].log_data[94].valid := 1, [26].log_data[95].valid := 1, [26].log_data[96].valid := 1, [26].log_data[97].valid := 1, [26].log_data[98].valid := 1, [26].log_data[99].valid := 1, [26].log_data[100].valid := 1, [26].log_data[101].valid := 1, [26].log_data[102].valid := 1, [26].log_data[103].valid := 1, [26].log_data[104].valid := 1, [26].log_data[105].valid := 1, [26].log_data[106].valid := 1, [26].log_data[107].valid := 1, [26].log_data[108].valid := 1, [26].log_data[109].valid := 1, [26].log_data[110].valid := 1, [26].log_data[111].valid := 1, [26].log_data[112].valid := 1, [26].log_data[113].valid := 1, [26].log_data[114].valid := 1, [26].log_data[115].valid := 1, [26].log_data[116].valid := 1, [26].log_data[117].valid := 1, [26].log_data[118].valid := 1, [26].log_data[119].valid := 1, [26].log_data[120].valid := 1, [26].log_data[121].valid := 1, [26].log_data[122].valid := 1, [26].log_data[123].valid := 1, [26].log_data[124].valid := 1, [26].time.Year := 2023, [26].time.Month := 1, [26].time.Day := 14, [26].time.Hour := 5, [26].time.Minute := 59, [26].time.Second := 59, [27].log_data[0].min := 1.0, [27].log_data[0].max := 1.0, [27].log_data[0].total := 3600.0, [27].log_data[0].time := 3600.0, [27].log_data[0].valid := 1, [27].log_data[1].max := 1.0, [27].log_data[1].total := 535.0, [27].log_data[1].time := 3600.0, [27].log_data[1].maxminute := 49, [27].log_data[1].valid := 1,
        [27].log_data[2].max := 1.0, [27].log_data[2].total := 531.5, [27].log_data[2].time := 3600.0, [27].log_data[2].maxminute := 49, [27].log_data[2].valid := 1, [27].log_data[3].time := 3600.0, [27].log_data[3].valid := 1, [27].log_data[4].time := 3600.0, [27].log_data[4].valid := 1, [27].log_data[5].max := 1.0, [27].log_data[5].total := 217.0, [27].log_data[5].time := 3600.0, [27].log_data[5].maxminute := 51, [27].log_data[5].valid := 1, [27].log_data[6].time := 3600.0, [27].log_data[6].valid := 1, [27].log_data[7].time := 3600.0, [27].log_data[7].valid := 1, [27].log_data[8].max := 1.0, [27].log_data[8].total := 401.749, [27].log_data[8].time := 3600.0, [27].log_data[8].maxminute := 53, [27].log_data[8].valid := 1, [27].log_data[9].max := 1.0, [27].log_data[9].total := 398.249, [27].log_data[9].time := 3600.0, [27].log_data[9].maxminute := 53, [27].log_data[9].valid := 1, [27].log_data[10].min := 1.0, [27].log_data[10].max := 1.0, [27].log_data[10].total := 3600.0, [27].log_data[10].time := 3600.0, [27].log_data[10].valid := 1, [27].log_data[11].time := 3600.0, [27].log_data[11].valid := 1, [27].log_data[12].min := 1.0, [27].log_data[12].max := 1.0, [27].log_data[12].total := 3600.0, [27].log_data[12].time := 3600.0, [27].log_data[12].valid := 1, [27].log_data[13].min := 1.0, [27].log_data[13].max := 1.0, [27].log_data[13].total := 3600.0, [27].log_data[13].time := 3600.0, [27].log_data[13].valid := 1, [27].log_data[14].time := 3600.0, [27].log_data[14].valid := 1, [27].log_data[15].time := 3600.0, [27].log_data[15].valid := 1, [27].log_data[16].time := 3600.0, [27].log_data[16].valid := 1, [27].log_data[17].min := 1.0, [27].log_data[17].max := 1.0, [27].log_data[17].total := 3600.0, [27].log_data[17].time := 3600.0, [27].log_data[17].valid := 1, [27].log_data[18].time := 3600.0, [27].log_data[18].valid := 1, [27].log_data[19].time := 3600.0, [27].log_data[19].valid := 1,
        [27].log_data[20].time := 3600.0, [27].log_data[20].valid := 1, [27].log_data[21].min := 1.0, [27].log_data[21].max := 1.0, [27].log_data[21].total := 3600.0, [27].log_data[21].time := 3600.0, [27].log_data[21].valid := 1, [27].log_data[22].time := 3600.0, [27].log_data[22].valid := 1, [27].log_data[23].time := 3600.0, [27].log_data[23].valid := 1, [27].log_data[24].time := 3600.0, [27].log_data[24].valid := 1, [27].log_data[25].time := 3600.0, [27].log_data[25].valid := 1, [27].log_data[26].time := 3600.0, [27].log_data[26].valid := 1, [27].log_data[27].time := 3600.0, [27].log_data[27].valid := 1, [27].log_data[28].time := 3600.0, [27].log_data[28].valid := 1, [27].log_data[29].min := 1.0, [27].log_data[29].max := 1.0, [27].log_data[29].total := 3600.0, [27].log_data[29].time := 3600.0, [27].log_data[29].valid := 1, [27].log_data[30].min := 1.0, [27].log_data[30].max := 1.0, [27].log_data[30].total := 3600.0, [27].log_data[30].time := 3600.0, [27].log_data[30].valid := 1, [27].log_data[31].time := 3600.0, [27].log_data[31].valid := 1, [27].log_data[32].max := 1.0, [27].log_data[32].total := 394.749, [27].log_data[32].time := 3600.0, [27].log_data[32].maxminute := 53, [27].log_data[32].valid := 1, [27].log_data[33].time := 3600.0, [27].log_data[33].valid := 1, [27].log_data[34].time := 3600.0, [27].log_data[34].valid := 1, [27].log_data[35].max := 1.0, [27].log_data[35].total := 130.249, [27].log_data[35].time := 3600.0, [27].log_data[35].maxminute := 57, [27].log_data[35].valid := 1, [27].log_data[36].max := 1.0, [27].log_data[36].total := 172.749, [27].log_data[36].time := 3600.0, [27].log_data[36].maxminute := 53, [27].log_data[36].valid := 1, [27].log_data[37].max := 7.3455496, [27].log_data[37].total := 3398.4998, [27].log_data[37].time := 3600.0, [27].log_data[37].maxminute := 50, [27].log_data[37].valid := 1, [27].log_data[38].time := 3600.0, [27].log_data[38].valid := 1, [27].log_data[39].min := 0.9941174,
        [27].log_data[39].max := 1.0221478, [27].log_data[39].total := 3610.1514, [27].log_data[39].time := 3600.0, [27].log_data[39].minminute := 40, [27].log_data[39].maxminute := 55, [27].log_data[39].valid := 1, [27].log_data[40].min := 7.553049, [27].log_data[40].max := 7.599217, [27].log_data[40].total := 27286.537, [27].log_data[40].time := 3600.0, [27].log_data[40].minminute := 31, [27].log_data[40].maxminute := 58, [27].log_data[40].valid := 1, [27].log_data[41].min := 0.040795166, [27].log_data[41].max := 0.05767627, [27].log_data[41].total := 168.36761, [27].log_data[41].time := 3600.0, [27].log_data[41].minminute := 39, [27].log_data[41].maxminute := 7, [27].log_data[41].valid := 1, [27].log_data[42].min := 2.2928205, [27].log_data[42].max := 2.297296, [27].log_data[42].total := 8262.819, [27].log_data[42].time := 3600.0, [27].log_data[42].minminute := 5, [27].log_data[42].valid := 1, [27].log_data[43].min := -0.26000214, [27].log_data[43].max := -0.26000214, [27].log_data[43].total := -935.9732, [27].log_data[43].time := 3600.0, [27].log_data[43].valid := 1, [27].log_data[44].min := -0.30000305, [27].log_data[44].max := -0.27999878, [27].log_data[44].total := -1016.7734, [27].log_data[44].time := 3600.0, [27].log_data[44].valid := 1, [27].log_data[45].time := 3600.0, [27].log_data[45].valid := 1, [27].log_data[46].time := 3600.0, [27].log_data[46].valid := 1, [27].log_data[47].time := 3600.0, [27].log_data[47].valid := 1, [27].log_data[48].min := 6.7692976, [27].log_data[48].max := 6.9608383, [27].log_data[48].total := 24444.244, [27].log_data[48].time := 3600.0, [27].log_data[48].minminute := 1, [27].log_data[48].maxminute := 57, [27].log_data[48].valid := 1, [27].log_data[49].min := 8.49271, [27].log_data[49].max := 9.64494, [27].log_data[49].total := 34353.63, [27].log_data[49].time := 3600.0, [27].log_data[49].minminute := 59, [27].log_data[49].maxminute := 41, [27].log_data[49].valid := 1, [27].log_data[50].min := 2.0616283, [27].log_data[50].max := 2.1520796, [27].log_data[50].total := 7588.832, [27].log_data[50].time := 3600.0,
        [27].log_data[50].minminute := 55, [27].log_data[50].maxminute := 53, [27].log_data[50].valid := 1, [27].log_data[51].time := 3600.0, [27].log_data[51].valid := 1, [27].log_data[52].min := -4.2599945, [27].log_data[52].max := -1.4800034, [27].log_data[52].total := -6036.944, [27].log_data[52].time := 3600.0, [27].log_data[52].minminute := 53, [27].log_data[52].maxminute := 10, [27].log_data[52].valid := 1, [27].log_data[53].min := -4.0199966, [27].log_data[53].max := 0.22000122, [27].log_data[53].total := -5556.235, [27].log_data[53].time := 3600.0, [27].log_data[53].minminute := 53, [27].log_data[53].maxminute := 57, [27].log_data[53].valid := 1, [27].log_data[54].max := 0.534, [27].log_data[54].total := 155.67178, [27].log_data[54].time := 3600.0, [27].log_data[54].maxminute := 53, [27].log_data[54].valid := 1, [27].log_data[55].max := 0.4965, [27].log_data[55].total := 117.141945, [27].log_data[55].time := 3600.0, [27].log_data[55].maxminute := 57, [27].log_data[55].valid := 1, [27].log_data[56].min := 0.16036338, [27].log_data[56].max := 0.16075596, [27].log_data[56].total := 577.7974, [27].log_data[56].time := 3600.0, [27].log_data[56].minminute := 3, [27].log_data[56].maxminute := 38, [27].log_data[56].valid := 1, [27].log_data[57].min := 0.30094728, [27].log_data[57].max := 0.3013791, [27].log_data[57].total := 1083.953, [27].log_data[57].time := 3600.0, [27].log_data[57].minminute := 1, [27].log_data[57].maxminute := 13, [27].log_data[57].valid := 1, [27].log_data[58].time := 3600.0, [27].log_data[58].valid := 1, [27].log_data[59].time := 3600.0, [27].log_data[59].valid := 1, [27].log_data[60].valid := 1, [27].log_data[61].valid := 1, [27].log_data[62].valid := 1, [27].log_data[63].valid := 1, [27].log_data[64].valid := 1, [27].log_data[65].valid := 1, [27].log_data[66].valid := 1, [27].log_data[67].valid := 1, [27].log_data[68].valid := 1, [27].log_data[69].valid := 1, [27].log_data[70].valid := 1, [27].log_data[71].valid := 1, [27].log_data[72].valid := 1,
        [27].log_data[73].valid := 1, [27].log_data[74].valid := 1, [27].log_data[75].valid := 1, [27].log_data[76].valid := 1, [27].log_data[77].valid := 1, [27].log_data[78].valid := 1, [27].log_data[79].valid := 1, [27].log_data[80].valid := 1, [27].log_data[81].valid := 1, [27].log_data[82].valid := 1, [27].log_data[83].valid := 1, [27].log_data[84].valid := 1, [27].log_data[85].valid := 1, [27].log_data[86].valid := 1, [27].log_data[87].valid := 1, [27].log_data[88].valid := 1, [27].log_data[89].valid := 1, [27].log_data[90].valid := 1, [27].log_data[91].valid := 1, [27].log_data[92].valid := 1, [27].log_data[93].valid := 1, [27].log_data[94].valid := 1, [27].log_data[95].valid := 1, [27].log_data[96].valid := 1, [27].log_data[97].valid := 1, [27].log_data[98].valid := 1, [27].log_data[99].valid := 1, [27].log_data[100].valid := 1, [27].log_data[101].valid := 1, [27].log_data[102].valid := 1, [27].log_data[103].valid := 1, [27].log_data[104].valid := 1, [27].log_data[105].valid := 1, [27].log_data[106].valid := 1, [27].log_data[107].valid := 1, [27].log_data[108].valid := 1, [27].log_data[109].valid := 1, [27].log_data[110].valid := 1, [27].log_data[111].valid := 1, [27].log_data[112].valid := 1, [27].log_data[113].valid := 1, [27].log_data[114].valid := 1, [27].log_data[115].valid := 1, [27].log_data[116].valid := 1, [27].log_data[117].valid := 1, [27].log_data[118].valid := 1, [27].log_data[119].valid := 1, [27].log_data[120].valid := 1, [27].log_data[121].valid := 1, [27].log_data[122].valid := 1, [27].log_data[123].valid := 1, [27].log_data[124].valid := 1, [27].time.Year := 2023, [27].time.Month := 1, [27].time.Day := 14, [27].time.Hour := 6, [27].time.Minute := 59, [27].time.Second := 59, [28].log_data[0].min := 1.0, [28].log_data[0].max := 1.0,
        [28].log_data[0].total := 3600.0, [28].log_data[0].time := 3600.0, [28].log_data[0].valid := 1, [28].log_data[1].time := 3600.0, [28].log_data[1].valid := 1, [28].log_data[2].time := 3600.0, [28].log_data[2].valid := 1, [28].log_data[3].time := 3600.0, [28].log_data[3].valid := 1, [28].log_data[4].time := 3600.0, [28].log_data[4].valid := 1, [28].log_data[5].time := 3600.0, [28].log_data[5].valid := 1, [28].log_data[6].time := 3600.0, [28].log_data[6].valid := 1, [28].log_data[7].time := 3600.0, [28].log_data[7].valid := 1, [28].log_data[8].min := 1.0, [28].log_data[8].max := 1.0, [28].log_data[8].total := 3600.0, [28].log_data[8].time := 3600.0, [28].log_data[8].valid := 1, [28].log_data[9].min := 1.0, [28].log_data[9].max := 1.0, [28].log_data[9].total := 3600.0, [28].log_data[9].time := 3600.0, [28].log_data[9].valid := 1, [28].log_data[10].min := 1.0, [28].log_data[10].max := 1.0, [28].log_data[10].total := 3600.0, [28].log_data[10].time := 3600.0, [28].log_data[10].valid := 1, [28].log_data[11].time := 3600.0, [28].log_data[11].valid := 1, [28].log_data[12].min := 1.0, [28].log_data[12].max := 1.0, [28].log_data[12].total := 3600.0, [28].log_data[12].time := 3600.0, [28].log_data[12].valid := 1, [28].log_data[13].min := 1.0, [28].log_data[13].max := 1.0, [28].log_data[13].total := 3600.0, [28].log_data[13].time := 3600.0, [28].log_data[13].valid := 1, [28].log_data[14].time := 3600.0, [28].log_data[14].valid := 1, [28].log_data[15].time := 3600.0, [28].log_data[15].valid := 1, [28].log_data[16].time := 3600.0, [28].log_data[16].valid := 1, [28].log_data[17].min := 1.0, [28].log_data[17].max := 1.0, [28].log_data[17].total := 3600.0, [28].log_data[17].time := 3600.0, [28].log_data[17].valid := 1, [28].log_data[18].time := 3600.0, [28].log_data[18].valid := 1, [28].log_data[19].time := 3600.0, [28].log_data[19].valid := 1, [28].log_data[20].time := 3600.0,
        [28].log_data[20].valid := 1, [28].log_data[21].min := 1.0, [28].log_data[21].max := 1.0, [28].log_data[21].total := 3600.0, [28].log_data[21].time := 3600.0, [28].log_data[21].valid := 1, [28].log_data[22].time := 3600.0, [28].log_data[22].valid := 1, [28].log_data[23].time := 3600.0, [28].log_data[23].valid := 1, [28].log_data[24].time := 3600.0, [28].log_data[24].valid := 1, [28].log_data[25].time := 3600.0, [28].log_data[25].valid := 1, [28].log_data[26].time := 3600.0, [28].log_data[26].valid := 1, [28].log_data[27].time := 3600.0, [28].log_data[27].valid := 1, [28].log_data[28].time := 3600.0, [28].log_data[28].valid := 1, [28].log_data[29].min := 1.0, [28].log_data[29].max := 1.0, [28].log_data[29].total := 3600.0, [28].log_data[29].time := 3600.0, [28].log_data[29].valid := 1, [28].log_data[30].min := 1.0, [28].log_data[30].max := 1.0, [28].log_data[30].total := 3600.0, [28].log_data[30].time := 3600.0, [28].log_data[30].valid := 1, [28].log_data[31].max := 1.0, [28].log_data[31].total := 1629.7471, [28].log_data[31].time := 3600.0, [28].log_data[31].maxminute := 3, [28].log_data[31].valid := 1, [28].log_data[32].max := 1.0, [28].log_data[32].total := 1440.998, [28].log_data[32].time := 3600.0, [28].log_data[32].minminute := 1, [28].log_data[32].valid := 1, [28].log_data[33].time := 3600.0, [28].log_data[33].valid := 1, [28].log_data[34].time := 3600.0, [28].log_data[34].valid := 1, [28].log_data[35].max := 1.0, [28].log_data[35].total := 1499.498, [28].log_data[35].time := 3600.0, [28].log_data[35].minminute := 6, [28].log_data[35].valid := 1, [28].log_data[36].max := 1.0, [28].log_data[36].total := 1629.7471, [28].log_data[36].time := 3600.0, [28].log_data[36].maxminute := 8, [28].log_data[36].valid := 1, [28].log_data[37].time := 3600.0, [28].log_data[37].valid := 1, [28].log_data[38].time := 3600.0, [28].log_data[38].valid := 1, [28].log_data[39].min := 0.9976506, [28].log_data[39].max := 1.0098991,
        [28].log_data[39].total := 3616.6113, [28].log_data[39].time := 3600.0, [28].log_data[39].minminute := 29, [28].log_data[39].maxminute := 57, [28].log_data[39].valid := 1, [28].log_data[40].min := 7.5571713, [28].log_data[40].max := 7.5959196, [28].log_data[40].total := 27289.766, [28].log_data[40].time := 3600.0, [28].log_data[40].minminute := 24, [28].log_data[40].maxminute := 48, [28].log_data[40].valid := 1, [28].log_data[41].min := 0.025680907, [28].log_data[41].max := 0.052572753, [28].log_data[41].total := 131.85948, [28].log_data[41].time := 3600.0, [28].log_data[41].minminute := 36, [28].log_data[41].maxminute := 56, [28].log_data[41].valid := 1, [28].log_data[42].min := 2.292467, [28].log_data[42].max := 2.2974136, [28].log_data[42].total := 8262.718, [28].log_data[42].time := 3600.0, [28].log_data[42].minminute := 30, [28].log_data[42].maxminute := 3, [28].log_data[42].valid := 1, [28].log_data[43].min := -0.26000214, [28].log_data[43].max := -0.26000214, [28].log_data[43].total := -935.9732, [28].log_data[43].time := 3600.0, [28].log_data[43].valid := 1, [28].log_data[44].min := -0.30000305, [28].log_data[44].max := -0.27999878, [28].log_data[44].total := -1023.56726, [28].log_data[44].time := 3600.0, [28].log_data[44].valid := 1, [28].log_data[45].time := 3600.0, [28].log_data[45].valid := 1, [28].log_data[46].time := 3600.0, [28].log_data[46].valid := 1, [28].log_data[47].time := 3600.0, [28].log_data[47].valid := 1, [28].log_data[48].min := 6.595069, [28].log_data[48].max := 6.8407474, [28].log_data[48].total := 24190.197, [28].log_data[48].time := 3600.0, [28].log_data[48].minminute := 21, [28].log_data[48].valid := 1, [28].log_data[49].min := 7.1176887, [28].log_data[49].max := 9.539139, [28].log_data[49].total := 30107.92, [28].log_data[49].time := 3600.0, [28].log_data[49].minminute := 19, [28].log_data[49].maxminute := 59, [28].log_data[49].valid := 1, [28].log_data[50].min := 2.0061567, [28].log_data[50].max := 2.0997875, [28].log_data[50].total := 7415.8945, [28].log_data[50].time := 3600.0, [28].log_data[50].minminute := 59,
        [28].log_data[50].valid := 1, [28].log_data[51].time := 3600.0, [28].log_data[51].valid := 1, [28].log_data[52].min := -2.840004, [28].log_data[52].max := 0.11999512, [28].log_data[52].total := -7553.861, [28].log_data[52].time := 3600.0, [28].log_data[52].minminute := 24, [28].log_data[52].maxminute := 2, [28].log_data[52].valid := 1, [28].log_data[53].min := -2.4800034, [28].log_data[53].max := 0.22000122, [28].log_data[53].total := -7020.0, [28].log_data[53].time := 3600.0, [28].log_data[53].minminute := 48, [28].log_data[53].maxminute := 7, [28].log_data[53].valid := 1, [28].log_data[54].max := 0.514, [28].log_data[54].total := 1217.1643, [28].log_data[54].time := 3600.0, [28].log_data[54].minminute := 2, [28].log_data[54].maxminute := 56, [28].log_data[54].valid := 1, [28].log_data[55].max := 0.5105, [28].log_data[55].total := 1242.7908, [28].log_data[55].time := 3600.0, [28].log_data[55].minminute := 6, [28].log_data[55].maxminute := 50, [28].log_data[55].valid := 1, [28].log_data[56].min := 0.16032413, [28].log_data[56].max := 0.16075596, [28].log_data[56].total := 577.8137, [28].log_data[56].time := 3600.0, [28].log_data[56].minminute := 28, [28].log_data[56].maxminute := 36, [28].log_data[56].valid := 1, [28].log_data[57].min := 0.2993377, [28].log_data[57].max := 0.30133983, [28].log_data[57].total := 1080.6187, [28].log_data[57].time := 3600.0, [28].log_data[57].minminute := 30, [28].log_data[57].maxminute := 12, [28].log_data[57].valid := 1, [28].log_data[58].time := 3600.0, [28].log_data[58].valid := 1, [28].log_data[59].time := 3600.0, [28].log_data[59].valid := 1, [28].log_data[60].valid := 1, [28].log_data[61].valid := 1, [28].log_data[62].valid := 1, [28].log_data[63].valid := 1, [28].log_data[64].valid := 1, [28].log_data[65].valid := 1, [28].log_data[66].valid := 1, [28].log_data[67].valid := 1, [28].log_data[68].valid := 1, [28].log_data[69].valid := 1, [28].log_data[70].valid := 1, [28].log_data[71].valid := 1, [28].log_data[72].valid := 1,
        [28].log_data[73].valid := 1, [28].log_data[74].valid := 1, [28].log_data[75].valid := 1, [28].log_data[76].valid := 1, [28].log_data[77].valid := 1, [28].log_data[78].valid := 1, [28].log_data[79].valid := 1, [28].log_data[80].valid := 1, [28].log_data[81].valid := 1, [28].log_data[82].valid := 1, [28].log_data[83].valid := 1, [28].log_data[84].valid := 1, [28].log_data[85].valid := 1, [28].log_data[86].valid := 1, [28].log_data[87].valid := 1, [28].log_data[88].valid := 1, [28].log_data[89].valid := 1, [28].log_data[90].valid := 1, [28].log_data[91].valid := 1, [28].log_data[92].valid := 1, [28].log_data[93].valid := 1, [28].log_data[94].valid := 1, [28].log_data[95].valid := 1, [28].log_data[96].valid := 1, [28].log_data[97].valid := 1, [28].log_data[98].valid := 1, [28].log_data[99].valid := 1, [28].log_data[100].valid := 1, [28].log_data[101].valid := 1, [28].log_data[102].valid := 1, [28].log_data[103].valid := 1, [28].log_data[104].valid := 1, [28].log_data[105].valid := 1, [28].log_data[106].valid := 1, [28].log_data[107].valid := 1, [28].log_data[108].valid := 1, [28].log_data[109].valid := 1, [28].log_data[110].valid := 1, [28].log_data[111].valid := 1, [28].log_data[112].valid := 1, [28].log_data[113].valid := 1, [28].log_data[114].valid := 1, [28].log_data[115].valid := 1, [28].log_data[116].valid := 1, [28].log_data[117].valid := 1, [28].log_data[118].valid := 1, [28].log_data[119].valid := 1, [28].log_data[120].valid := 1, [28].log_data[121].valid := 1, [28].log_data[122].valid := 1, [28].log_data[123].valid := 1, [28].log_data[124].valid := 1, [28].time.Year := 2023, [28].time.Month := 1, [28].time.Day := 14, [28].time.Hour := 7, [28].time.Minute := 59, [28].time.Second := 59, [29].log_data[0].min := 1.0, [29].log_data[0].max := 1.0,
        [29].log_data[0].total := 3600.0, [29].log_data[0].time := 3600.0, [29].log_data[0].valid := 1, [29].log_data[1].time := 3600.0, [29].log_data[1].valid := 1, [29].log_data[2].time := 3600.0, [29].log_data[2].valid := 1, [29].log_data[3].time := 3600.0, [29].log_data[3].valid := 1, [29].log_data[4].time := 3600.0, [29].log_data[4].valid := 1, [29].log_data[5].time := 3600.0, [29].log_data[5].valid := 1, [29].log_data[6].time := 3600.0, [29].log_data[6].valid := 1, [29].log_data[7].time := 3600.0, [29].log_data[7].valid := 1, [29].log_data[8].max := 1.0, [29].log_data[8].total := 139.751, [29].log_data[8].time := 3600.0, [29].log_data[8].minminute := 2, [29].log_data[8].valid := 1, [29].log_data[9].max := 1.0, [29].log_data[9].total := 139.751, [29].log_data[9].time := 3600.0, [29].log_data[9].minminute := 2, [29].log_data[9].valid := 1, [29].log_data[10].min := 1.0, [29].log_data[10].max := 1.0, [29].log_data[10].total := 3600.0, [29].log_data[10].time := 3600.0, [29].log_data[10].valid := 1, [29].log_data[11].time := 3600.0, [29].log_data[11].valid := 1, [29].log_data[12].min := 1.0, [29].log_data[12].max := 1.0, [29].log_data[12].total := 3600.0, [29].log_data[12].time := 3600.0, [29].log_data[12].valid := 1, [29].log_data[13].min := 1.0, [29].log_data[13].max := 1.0, [29].log_data[13].total := 3600.0, [29].log_data[13].time := 3600.0, [29].log_data[13].valid := 1, [29].log_data[14].time := 3600.0, [29].log_data[14].valid := 1, [29].log_data[15].time := 3600.0, [29].log_data[15].valid := 1, [29].log_data[16].time := 3600.0, [29].log_data[16].valid := 1, [29].log_data[17].min := 1.0, [29].log_data[17].max := 1.0, [29].log_data[17].total := 3600.0, [29].log_data[17].time := 3600.0, [29].log_data[17].valid := 1, [29].log_data[18].time := 3600.0, [29].log_data[18].valid := 1, [29].log_data[19].time := 3600.0, [29].log_data[19].valid := 1, [29].log_data[20].time := 3600.0,
        [29].log_data[20].valid := 1, [29].log_data[21].min := 1.0, [29].log_data[21].max := 1.0, [29].log_data[21].total := 3600.0, [29].log_data[21].time := 3600.0, [29].log_data[21].valid := 1, [29].log_data[22].time := 3600.0, [29].log_data[22].valid := 1, [29].log_data[23].time := 3600.0, [29].log_data[23].valid := 1, [29].log_data[24].time := 3600.0, [29].log_data[24].valid := 1, [29].log_data[25].time := 3600.0, [29].log_data[25].valid := 1, [29].log_data[26].time := 3600.0, [29].log_data[26].valid := 1, [29].log_data[27].time := 3600.0, [29].log_data[27].valid := 1, [29].log_data[28].time := 3600.0, [29].log_data[28].valid := 1, [29].log_data[29].min := 1.0, [29].log_data[29].max := 1.0, [29].log_data[29].total := 3600.0, [29].log_data[29].time := 3600.0, [29].log_data[29].valid := 1, [29].log_data[30].min := 1.0, [29].log_data[30].max := 1.0, [29].log_data[30].total := 3600.0, [29].log_data[30].time := 3600.0, [29].log_data[30].valid := 1, [29].log_data[31].time := 3600.0, [29].log_data[31].valid := 1, [29].log_data[32].max := 1.0, [29].log_data[32].total := 143.5, [29].log_data[32].time := 3600.0, [29].log_data[32].minminute := 2, [29].log_data[32].valid := 1, [29].log_data[33].time := 3600.0, [29].log_data[33].valid := 1, [29].log_data[34].time := 3600.0, [29].log_data[34].valid := 1, [29].log_data[35].max := 1.0, [29].log_data[35].total := 84.749, [29].log_data[35].time := 3600.0, [29].log_data[35].valid := 1, [29].log_data[36].time := 3600.0, [29].log_data[36].valid := 1, [29].log_data[37].time := 3600.0, [29].log_data[37].valid := 1, [29].log_data[38].time := 3600.0, [29].log_data[38].valid := 1, [29].log_data[39].min := 0.99788606, [29].log_data[39].max := 1.0101347, [29].log_data[39].total := 3617.055, [29].log_data[39].time := 3600.0, [29].log_data[39].minminute := 46, [29].log_data[39].maxminute := 50, [29].log_data[39].valid := 1, [29].log_data[40].min := 7.553049, [29].log_data[40].max := 7.589324,
        [29].log_data[40].total := 27292.24, [29].log_data[40].time := 3600.0, [29].log_data[40].minminute := 17, [29].log_data[40].maxminute := 20, [29].log_data[40].valid := 1, [29].log_data[41].min := 0.038832273, [29].log_data[41].max := 0.0535542, [29].log_data[41].total := 162.72957, [29].log_data[41].time := 3600.0, [29].log_data[41].minminute := 39, [29].log_data[41].maxminute := 23, [29].log_data[41].valid := 1, [29].log_data[42].min := 2.2922316, [29].log_data[42].max := 2.2974136, [29].log_data[42].total := 8262.543, [29].log_data[42].time := 3600.0, [29].log_data[42].minminute := 40, [29].log_data[42].maxminute := 17, [29].log_data[42].valid := 1, [29].log_data[43].min := -0.26000214, [29].log_data[43].max := -0.23999786, [29].log_data[43].total := -935.9482, [29].log_data[43].time := 3600.0, [29].log_data[43].maxminute := 12, [29].log_data[43].valid := 1, [29].log_data[44].min := -0.30000305, [29].log_data[44].max := -0.27999878, [29].log_data[44].total := -1008.34106, [29].log_data[44].time := 3600.0, [29].log_data[44].valid := 1, [29].log_data[45].time := 3600.0, [29].log_data[45].valid := 1, [29].log_data[46].time := 3600.0, [29].log_data[46].valid := 1, [29].log_data[47].time := 3600.0, [29].log_data[47].valid := 1, [29].log_data[48].min := 6.740717, [29].log_data[48].max := 6.752809, [29].log_data[48].total := 24287.232, [29].log_data[48].time := 3600.0, [29].log_data[48].minminute := 6, [29].log_data[48].maxminute := 52, [29].log_data[48].valid := 1, [29].log_data[49].min := 9.503218, [29].log_data[49].max := 9.624525, [29].log_data[49].total := 34466.926, [29].log_data[49].time := 3600.0, [29].log_data[49].maxminute := 55, [29].log_data[49].valid := 1, [29].log_data[50].min := 1.9963813, [29].log_data[50].max := 2.1183958, [29].log_data[50].total := 7580.0464, [29].log_data[50].time := 3600.0, [29].log_data[50].minminute := 2, [29].log_data[50].maxminute := 23, [29].log_data[50].valid := 1, [29].log_data[51].time := 3600.0, [29].log_data[51].valid := 1, [29].log_data[52].min := -2.600006, [29].log_data[52].max := -0.08000183,
        [29].log_data[52].total := -5389.309, [29].log_data[52].time := 3600.0, [29].log_data[52].minminute := 1, [29].log_data[52].maxminute := 2, [29].log_data[52].valid := 1, [29].log_data[53].min := -2.4400024, [29].log_data[53].max := 0.11999512, [29].log_data[53].total := -4886.7046, [29].log_data[53].time := 3600.0, [29].log_data[53].minminute := 2, [29].log_data[53].valid := 1, [29].log_data[54].max := 0.427, [29].log_data[54].total := 57.639957, [29].log_data[54].time := 3600.0, [29].log_data[54].minminute := 2, [29].log_data[54].valid := 1, [29].log_data[55].max := 0.4965, [29].log_data[55].total := 32.006157, [29].log_data[55].time := 3600.0, [29].log_data[55].maxminute := 1, [29].log_data[55].valid := 1, [29].log_data[56].min := 0.16036338, [29].log_data[56].max := 0.16075596, [29].log_data[56].total := 577.8507, [29].log_data[56].time := 3600.0, [29].log_data[56].minminute := 8, [29].log_data[56].maxminute := 41, [29].log_data[56].valid := 1, [29].log_data[57].min := 0.29929844, [29].log_data[57].max := 0.29976952, [29].log_data[57].total := 1078.2483, [29].log_data[57].time := 3600.0, [29].log_data[57].minminute := 8, [29].log_data[57].maxminute := 56, [29].log_data[57].valid := 1, [29].log_data[58].time := 3600.0, [29].log_data[58].valid := 1, [29].log_data[59].time := 3600.0, [29].log_data[59].valid := 1, [29].log_data[60].valid := 1, [29].log_data[61].valid := 1, [29].log_data[62].valid := 1, [29].log_data[63].valid := 1, [29].log_data[64].valid := 1, [29].log_data[65].valid := 1, [29].log_data[66].valid := 1, [29].log_data[67].valid := 1, [29].log_data[68].valid := 1, [29].log_data[69].valid := 1, [29].log_data[70].valid := 1, [29].log_data[71].valid := 1, [29].log_data[72].valid := 1, [29].log_data[73].valid := 1, [29].log_data[74].valid := 1, [29].log_data[75].valid := 1, [29].log_data[76].valid := 1, [29].log_data[77].valid := 1, [29].log_data[78].valid := 1, [29].log_data[79].valid := 1, [29].log_data[80].valid := 1,
        [29].log_data[81].valid := 1, [29].log_data[82].valid := 1, [29].log_data[83].valid := 1, [29].log_data[84].valid := 1, [29].log_data[85].valid := 1, [29].log_data[86].valid := 1, [29].log_data[87].valid := 1, [29].log_data[88].valid := 1, [29].log_data[89].valid := 1, [29].log_data[90].valid := 1, [29].log_data[91].valid := 1, [29].log_data[92].valid := 1, [29].log_data[93].valid := 1, [29].log_data[94].valid := 1, [29].log_data[95].valid := 1, [29].log_data[96].valid := 1, [29].log_data[97].valid := 1, [29].log_data[98].valid := 1, [29].log_data[99].valid := 1, [29].log_data[100].valid := 1, [29].log_data[101].valid := 1, [29].log_data[102].valid := 1, [29].log_data[103].valid := 1, [29].log_data[104].valid := 1, [29].log_data[105].valid := 1, [29].log_data[106].valid := 1, [29].log_data[107].valid := 1, [29].log_data[108].valid := 1, [29].log_data[109].valid := 1, [29].log_data[110].valid := 1, [29].log_data[111].valid := 1, [29].log_data[112].valid := 1, [29].log_data[113].valid := 1, [29].log_data[114].valid := 1, [29].log_data[115].valid := 1, [29].log_data[116].valid := 1, [29].log_data[117].valid := 1, [29].log_data[118].valid := 1, [29].log_data[119].valid := 1, [29].log_data[120].valid := 1, [29].log_data[121].valid := 1, [29].log_data[122].valid := 1, [29].log_data[123].valid := 1, [29].log_data[124].valid := 1, [29].time.Year := 2023, [29].time.Month := 1, [29].time.Day := 14, [29].time.Hour := 8, [29].time.Minute := 59, [29].time.Second := 59, [30].log_data[0].min := 1.0, [30].log_data[0].max := 1.0, [30].log_data[0].total := 3600.0, [30].log_data[0].time := 3600.0, [30].log_data[0].valid := 1, [30].log_data[1].max := 1.0, [30].log_data[1].total := 556.0, [30].log_data[1].time := 3600.0, [30].log_data[1].maxminute := 29, [30].log_data[1].valid := 1,
        [30].log_data[2].max := 1.0, [30].log_data[2].total := 552.5, [30].log_data[2].time := 3600.0, [30].log_data[2].maxminute := 29, [30].log_data[2].valid := 1, [30].log_data[3].time := 3600.0, [30].log_data[3].valid := 1, [30].log_data[4].time := 3600.0, [30].log_data[4].valid := 1, [30].log_data[5].max := 1.0, [30].log_data[5].total := 238.5, [30].log_data[5].time := 3600.0, [30].log_data[5].maxminute := 31, [30].log_data[5].valid := 1, [30].log_data[6].time := 3600.0, [30].log_data[6].valid := 1, [30].log_data[7].time := 3600.0, [30].log_data[7].valid := 1, [30].log_data[8].max := 1.0, [30].log_data[8].total := 1656.749, [30].log_data[8].time := 3600.0, [30].log_data[8].maxminute := 32, [30].log_data[8].valid := 1, [30].log_data[9].max := 1.0, [30].log_data[9].total := 1653.249, [30].log_data[9].time := 3600.0, [30].log_data[9].maxminute := 32, [30].log_data[9].valid := 1, [30].log_data[10].min := 1.0, [30].log_data[10].max := 1.0, [30].log_data[10].total := 3600.0, [30].log_data[10].time := 3600.0, [30].log_data[10].valid := 1, [30].log_data[11].time := 3600.0, [30].log_data[11].valid := 1, [30].log_data[12].min := 1.0, [30].log_data[12].max := 1.0, [30].log_data[12].total := 3600.0, [30].log_data[12].time := 3600.0, [30].log_data[12].valid := 1, [30].log_data[13].min := 1.0, [30].log_data[13].max := 1.0, [30].log_data[13].total := 3600.0, [30].log_data[13].time := 3600.0, [30].log_data[13].valid := 1, [30].log_data[14].time := 3600.0, [30].log_data[14].valid := 1, [30].log_data[15].time := 3600.0, [30].log_data[15].valid := 1, [30].log_data[16].time := 3600.0, [30].log_data[16].valid := 1, [30].log_data[17].min := 1.0, [30].log_data[17].max := 1.0, [30].log_data[17].total := 3600.0, [30].log_data[17].time := 3600.0, [30].log_data[17].valid := 1, [30].log_data[18].time := 3600.0, [30].log_data[18].valid := 1, [30].log_data[19].time := 3600.0, [30].log_data[19].valid := 1,
        [30].log_data[20].time := 3600.0, [30].log_data[20].valid := 1, [30].log_data[21].min := 1.0, [30].log_data[21].max := 1.0, [30].log_data[21].total := 3600.0, [30].log_data[21].time := 3600.0, [30].log_data[21].valid := 1, [30].log_data[22].time := 3600.0, [30].log_data[22].valid := 1, [30].log_data[23].time := 3600.0, [30].log_data[23].valid := 1, [30].log_data[24].time := 3600.0, [30].log_data[24].valid := 1, [30].log_data[25].time := 3600.0, [30].log_data[25].valid := 1, [30].log_data[26].time := 3600.0, [30].log_data[26].valid := 1, [30].log_data[27].time := 3600.0, [30].log_data[27].valid := 1, [30].log_data[28].time := 3600.0, [30].log_data[28].valid := 1, [30].log_data[29].min := 1.0, [30].log_data[29].max := 1.0, [30].log_data[29].total := 3600.0, [30].log_data[29].time := 3600.0, [30].log_data[29].valid := 1, [30].log_data[30].min := 1.0, [30].log_data[30].max := 1.0, [30].log_data[30].total := 3600.0, [30].log_data[30].time := 3600.0, [30].log_data[30].valid := 1, [30].log_data[31].max := 1.0, [30].log_data[31].total := 707.5, [30].log_data[31].time := 3600.0, [30].log_data[31].maxminute := 32, [30].log_data[31].valid := 1, [30].log_data[32].max := 1.0, [30].log_data[32].total := 677.49805, [30].log_data[32].time := 3600.0, [30].log_data[32].maxminute := 36, [30].log_data[32].valid := 1, [30].log_data[33].time := 3600.0, [30].log_data[33].valid := 1, [30].log_data[34].time := 3600.0, [30].log_data[34].valid := 1, [30].log_data[35].max := 1.0, [30].log_data[35].total := 543.249, [30].log_data[35].time := 3600.0, [30].log_data[35].maxminute := 41, [30].log_data[35].valid := 1, [30].log_data[36].max := 1.0, [30].log_data[36].total := 926.249, [30].log_data[36].time := 3600.0, [30].log_data[36].maxminute := 32, [30].log_data[36].valid := 1, [30].log_data[37].max := 7.5422335, [30].log_data[37].total := 3633.545, [30].log_data[37].time := 3600.0, [30].log_data[37].maxminute := 30, [30].log_data[37].valid := 1,
        [30].log_data[38].time := 3600.0, [30].log_data[38].valid := 1, [30].log_data[39].min := 0.9971795, [30].log_data[39].max := 1.0210879, [30].log_data[39].total := 3620.92, [30].log_data[39].time := 3600.0, [30].log_data[39].minminute := 37, [30].log_data[39].maxminute := 34, [30].log_data[39].valid := 1, [30].log_data[40].min := 7.558545, [30].log_data[40].max := 7.593171, [30].log_data[40].total := 27291.521, [30].log_data[40].time := 3600.0, [30].log_data[40].minminute := 35, [30].log_data[40].maxminute := 41, [30].log_data[40].valid := 1, [30].log_data[41].min := 0.046291504, [30].log_data[41].max := 0.06984644, [30].log_data[41].total := 215.69397, [30].log_data[41].time := 3600.0, [30].log_data[41].minminute := 35, [30].log_data[41].maxminute := 14, [30].log_data[41].valid := 1, [30].log_data[42].min := 2.2918782, [30].log_data[42].max := 2.2983558, [30].log_data[42].total := 8262.496, [30].log_data[42].time := 3600.0, [30].log_data[42].minminute := 47, [30].log_data[42].maxminute := 52, [30].log_data[42].valid := 1, [30].log_data[43].min := -0.26000214, [30].log_data[43].max := -0.23999786, [30].log_data[43].total := -935.8731, [30].log_data[43].time := 3600.0, [30].log_data[43].maxminute := 37, [30].log_data[43].valid := 1, [30].log_data[44].min := -0.30000305, [30].log_data[44].max := -0.27999878, [30].log_data[44].total := -1008.1059, [30].log_data[44].time := 3600.0, [30].log_data[44].minminute := 3, [30].log_data[44].valid := 1, [30].log_data[45].time := 3600.0, [30].log_data[45].valid := 1, [30].log_data[46].time := 3600.0, [30].log_data[46].valid := 1, [30].log_data[47].time := 3600.0, [30].log_data[47].valid := 1, [30].log_data[48].min := 6.585176, [30].log_data[48].max := 6.9591894, [30].log_data[48].total := 24292.44, [30].log_data[48].time := 3600.0, [30].log_data[48].minminute := 59, [30].log_data[48].maxminute := 37, [30].log_data[48].valid := 1, [30].log_data[49].min := 6.9802847, [30].log_data[49].max := 9.6500435, [30].log_data[49].total := 31700.705, [30].log_data[49].time := 3600.0, [30].log_data[49].minminute := 55,
        [30].log_data[49].maxminute := 19, [30].log_data[49].valid := 1, [30].log_data[50].min := 2.0545619, [30].log_data[50].max := 2.1505485, [30].log_data[50].total := 7588.6064, [30].log_data[50].time := 3600.0, [30].log_data[50].minminute := 34, [30].log_data[50].maxminute := 32, [30].log_data[50].valid := 1, [30].log_data[51].time := 3600.0, [30].log_data[51].valid := 1, [30].log_data[52].min := -4.4000015, [30].log_data[52].max := 0.13999939, [30].log_data[52].total := -6493.5103, [30].log_data[52].time := 3600.0, [30].log_data[52].minminute := 32, [30].log_data[52].maxminute := 56, [30].log_data[52].valid := 1, [30].log_data[53].min := -4.119995, [30].log_data[53].max := 0.2400055, [30].log_data[53].total := -6151.1157, [30].log_data[53].time := 3600.0, [30].log_data[53].minminute := 32, [30].log_data[53].maxminute := 41, [30].log_data[53].valid := 1, [30].log_data[54].max := 0.532, [30].log_data[54].total := 546.5264, [30].log_data[54].time := 3600.0, [30].log_data[54].maxminute := 36, [30].log_data[54].valid := 1, [30].log_data[55].max := 0.508, [30].log_data[55].total := 581.746, [30].log_data[55].time := 3600.0, [30].log_data[55].maxminute := 32, [30].log_data[55].valid := 1, [30].log_data[56].min := 0.16028486, [30].log_data[56].max := 0.16075596, [30].log_data[56].total := 577.7941, [30].log_data[56].time := 3600.0, [30].log_data[56].minminute := 59, [30].log_data[56].valid := 1, [30].log_data[57].min := 0.2991414, [30].log_data[57].max := 0.2998088, [30].log_data[57].total := 1078.4183, [30].log_data[57].time := 3600.0, [30].log_data[57].minminute := 59, [30].log_data[57].maxminute := 10, [30].log_data[57].valid := 1, [30].log_data[58].time := 3600.0, [30].log_data[58].valid := 1, [30].log_data[59].time := 3600.0, [30].log_data[59].valid := 1, [30].log_data[60].valid := 1, [30].log_data[61].valid := 1, [30].log_data[62].valid := 1, [30].log_data[63].valid := 1, [30].log_data[64].valid := 1, [30].log_data[65].valid := 1, [30].log_data[66].valid := 1, [30].log_data[67].valid := 1,
        [30].log_data[68].valid := 1, [30].log_data[69].valid := 1, [30].log_data[70].valid := 1, [30].log_data[71].valid := 1, [30].log_data[72].valid := 1, [30].log_data[73].valid := 1, [30].log_data[74].valid := 1, [30].log_data[75].valid := 1, [30].log_data[76].valid := 1, [30].log_data[77].valid := 1, [30].log_data[78].valid := 1, [30].log_data[79].valid := 1, [30].log_data[80].valid := 1, [30].log_data[81].valid := 1, [30].log_data[82].valid := 1, [30].log_data[83].valid := 1, [30].log_data[84].valid := 1, [30].log_data[85].valid := 1, [30].log_data[86].valid := 1, [30].log_data[87].valid := 1, [30].log_data[88].valid := 1, [30].log_data[89].valid := 1, [30].log_data[90].valid := 1, [30].log_data[91].valid := 1, [30].log_data[92].valid := 1, [30].log_data[93].valid := 1, [30].log_data[94].valid := 1, [30].log_data[95].valid := 1, [30].log_data[96].valid := 1, [30].log_data[97].valid := 1, [30].log_data[98].valid := 1, [30].log_data[99].valid := 1, [30].log_data[100].valid := 1, [30].log_data[101].valid := 1, [30].log_data[102].valid := 1, [30].log_data[103].valid := 1, [30].log_data[104].valid := 1, [30].log_data[105].valid := 1, [30].log_data[106].valid := 1, [30].log_data[107].valid := 1, [30].log_data[108].valid := 1, [30].log_data[109].valid := 1, [30].log_data[110].valid := 1, [30].log_data[111].valid := 1, [30].log_data[112].valid := 1, [30].log_data[113].valid := 1, [30].log_data[114].valid := 1, [30].log_data[115].valid := 1, [30].log_data[116].valid := 1, [30].log_data[117].valid := 1, [30].log_data[118].valid := 1, [30].log_data[119].valid := 1, [30].log_data[120].valid := 1, [30].log_data[121].valid := 1, [30].log_data[122].valid := 1, [30].log_data[123].valid := 1, [30].log_data[124].valid := 1, [30].time.Year := 2023, [30].time.Month := 1, [30].time.Day := 14,
        [30].time.Hour := 9, [30].time.Minute := 59, [30].time.Second := 59, [31].log_data[0].min := 1.0, [31].log_data[0].max := 1.0, [31].log_data[0].total := 3600.0, [31].log_data[0].time := 3600.0, [31].log_data[0].valid := 1, [31].log_data[1].max := 1.0, [31].log_data[1].total := 571.0, [31].log_data[1].time := 3600.0, [31].log_data[1].maxminute := 38, [31].log_data[1].valid := 1, [31].log_data[2].max := 1.0, [31].log_data[2].total := 567.5, [31].log_data[2].time := 3600.0, [31].log_data[2].maxminute := 38, [31].log_data[2].valid := 1, [31].log_data[3].time := 3600.0, [31].log_data[3].valid := 1, [31].log_data[4].time := 3600.0, [31].log_data[4].valid := 1, [31].log_data[5].max := 1.0, [31].log_data[5].total := 234.0, [31].log_data[5].time := 3600.0, [31].log_data[5].maxminute := 40, [31].log_data[5].valid := 1, [31].log_data[6].time := 3600.0, [31].log_data[6].valid := 1, [31].log_data[7].time := 3600.0, [31].log_data[7].valid := 1, [31].log_data[8].min := 1.0, [31].log_data[8].max := 1.0, [31].log_data[8].total := 3600.0, [31].log_data[8].time := 3600.0, [31].log_data[8].valid := 1, [31].log_data[9].min := 1.0, [31].log_data[9].max := 1.0, [31].log_data[9].total := 3600.0, [31].log_data[9].time := 3600.0, [31].log_data[9].valid := 1, [31].log_data[10].min := 1.0, [31].log_data[10].max := 1.0, [31].log_data[10].total := 3600.0, [31].log_data[10].time := 3600.0, [31].log_data[10].valid := 1, [31].log_data[11].time := 3600.0, [31].log_data[11].valid := 1, [31].log_data[12].min := 1.0, [31].log_data[12].max := 1.0, [31].log_data[12].total := 3600.0, [31].log_data[12].time := 3600.0, [31].log_data[12].valid := 1, [31].log_data[13].min := 1.0, [31].log_data[13].max := 1.0, [31].log_data[13].total := 3600.0, [31].log_data[13].time := 3600.0, [31].log_data[13].valid := 1, [31].log_data[14].time := 3600.0, [31].log_data[14].valid := 1,
        [31].log_data[15].time := 3600.0, [31].log_data[15].valid := 1, [31].log_data[16].time := 3600.0, [31].log_data[16].valid := 1, [31].log_data[17].min := 1.0, [31].log_data[17].max := 1.0, [31].log_data[17].total := 3600.0, [31].log_data[17].time := 3600.0, [31].log_data[17].valid := 1, [31].log_data[18].time := 3600.0, [31].log_data[18].valid := 1, [31].log_data[19].time := 3600.0, [31].log_data[19].valid := 1, [31].log_data[20].time := 3600.0, [31].log_data[20].valid := 1, [31].log_data[21].min := 1.0, [31].log_data[21].max := 1.0, [31].log_data[21].total := 3600.0, [31].log_data[21].time := 3600.0, [31].log_data[21].valid := 1, [31].log_data[22].time := 3600.0, [31].log_data[22].valid := 1, [31].log_data[23].time := 3600.0, [31].log_data[23].valid := 1, [31].log_data[24].time := 3600.0, [31].log_data[24].valid := 1, [31].log_data[25].time := 3600.0, [31].log_data[25].valid := 1, [31].log_data[26].time := 3600.0, [31].log_data[26].valid := 1, [31].log_data[27].time := 3600.0, [31].log_data[27].valid := 1, [31].log_data[28].time := 3600.0, [31].log_data[28].valid := 1, [31].log_data[29].min := 1.0, [31].log_data[29].max := 1.0, [31].log_data[29].total := 3600.0, [31].log_data[29].time := 3600.0, [31].log_data[29].valid := 1, [31].log_data[30].min := 1.0, [31].log_data[30].max := 1.0, [31].log_data[30].total := 3600.0, [31].log_data[30].time := 3600.0, [31].log_data[30].valid := 1, [31].log_data[31].max := 1.0, [31].log_data[31].total := 1629.7471, [31].log_data[31].time := 3600.0, [31].log_data[31].maxminute := 8, [31].log_data[31].valid := 1, [31].log_data[32].max := 1.0, [31].log_data[32].total := 1495.498, [31].log_data[32].time := 3600.0, [31].log_data[32].minminute := 6, [31].log_data[32].valid := 1, [31].log_data[33].time := 3600.0, [31].log_data[33].valid := 1, [31].log_data[34].time := 3600.0, [31].log_data[34].valid := 1, [31].log_data[35].max := 1.0, [31].log_data[35].total := 1629.7471,
        [31].log_data[35].time := 3600.0, [31].log_data[35].maxminute := 2, [31].log_data[35].valid := 1, [31].log_data[36].max := 1.0, [31].log_data[36].total := 1440.998, [31].log_data[36].time := 3600.0, [31].log_data[36].minminute := 1, [31].log_data[36].valid := 1, [31].log_data[37].max := 7.348298, [31].log_data[37].total := 3659.2856, [31].log_data[37].time := 3600.0, [31].log_data[37].maxminute := 39, [31].log_data[37].valid := 1, [31].log_data[38].time := 3600.0, [31].log_data[38].valid := 1, [31].log_data[39].min := 0.9970617, [31].log_data[39].max := 1.0225011, [31].log_data[39].total := 3626.4587, [31].log_data[39].time := 3600.0, [31].log_data[39].minminute := 42, [31].log_data[39].maxminute := 40, [31].log_data[39].valid := 1, [31].log_data[40].min := 7.5459046, [31].log_data[40].max := 7.600591, [31].log_data[40].total := 27289.79, [31].log_data[40].time := 3600.0, [31].log_data[40].minminute := 24, [31].log_data[40].maxminute := 30, [31].log_data[40].valid := 1, [31].log_data[41].min := 0.042169187, [31].log_data[41].max := 0.06356494, [31].log_data[41].total := 181.1406, [31].log_data[41].time := 3600.0, [31].log_data[41].minminute := 19, [31].log_data[41].valid := 1, [31].log_data[42].min := 2.292467, [31].log_data[42].max := 2.2970603, [31].log_data[42].total := 8262.289, [31].log_data[42].time := 3600.0, [31].log_data[42].minminute := 17, [31].log_data[42].maxminute := 4, [31].log_data[42].valid := 1, [31].log_data[43].min := -0.26000214, [31].log_data[43].max := -0.23999786, [31].log_data[43].total := -934.7641, [31].log_data[43].time := 3600.0, [31].log_data[43].maxminute := 1, [31].log_data[43].valid := 1, [31].log_data[44].min := -0.30000305, [31].log_data[44].max := -0.27999878, [31].log_data[44].total := -1007.8966, [31].log_data[44].time := 3600.0, [31].log_data[44].minminute := 35, [31].log_data[44].valid := 1, [31].log_data[45].time := 3600.0, [31].log_data[45].valid := 1, [31].log_data[46].time := 3600.0, [31].log_data[46].valid := 1, [31].log_data[47].time := 3600.0, [31].log_data[47].valid := 1,
        [31].log_data[48].min := 6.578031, [31].log_data[48].max := 6.9789753, [31].log_data[48].total := 24315.135, [31].log_data[48].time := 3600.0, [31].log_data[48].minminute := 1, [31].log_data[48].maxminute := 46, [31].log_data[48].valid := 1, [31].log_data[49].min := 7.0362277, [31].log_data[49].max := 9.535018, [31].log_data[49].total := 30509.217, [31].log_data[49].time := 3600.0, [31].log_data[49].maxminute := 40, [31].log_data[49].valid := 1, [31].log_data[50].min := 2.029947, [31].log_data[50].max := 2.1408908, [31].log_data[50].total := 7492.2495, [31].log_data[50].time := 3600.0, [31].log_data[50].minminute := 39, [31].log_data[50].maxminute := 46, [31].log_data[50].valid := 1, [31].log_data[51].time := 3600.0, [31].log_data[51].valid := 1, [31].log_data[52].min := -2.840004, [31].log_data[52].max := 0.13999939, [31].log_data[52].total := -7622.1816, [31].log_data[52].time := 3600.0, [31].log_data[52].minminute := 39, [31].log_data[52].maxminute := 6, [31].log_data[52].valid := 1, [31].log_data[53].min := -2.5600052, [31].log_data[53].max := 0.22000122, [31].log_data[53].total := -6828.0347, [31].log_data[53].time := 3600.0, [31].log_data[53].minminute := 44, [31].log_data[53].maxminute := 2, [31].log_data[53].valid := 1, [31].log_data[54].max := 0.5265, [31].log_data[54].total := 1241.3151, [31].log_data[54].time := 3600.0, [31].log_data[54].minminute := 6, [31].log_data[54].maxminute := 18, [31].log_data[54].valid := 1, [31].log_data[55].max := 0.534, [31].log_data[55].total := 1217.2072, [31].log_data[55].time := 3600.0, [31].log_data[55].minminute := 1, [31].log_data[55].maxminute := 23, [31].log_data[55].valid := 1, [31].log_data[56].min := 0.16028486, [31].log_data[56].max := 0.1607167, [31].log_data[56].total := 577.62286, [31].log_data[56].time := 3600.0, [31].log_data[56].maxminute := 40, [31].log_data[56].valid := 1, [31].log_data[57].min := 0.29757103, [31].log_data[57].max := 0.29937696, [31].log_data[57].total := 1072.2167, [31].log_data[57].time := 3600.0, [31].log_data[57].minminute := 10, [31].log_data[57].valid := 1,
        [31].log_data[58].time := 3600.0, [31].log_data[58].valid := 1, [31].log_data[59].time := 3600.0, [31].log_data[59].valid := 1, [31].log_data[60].valid := 1, [31].log_data[61].valid := 1, [31].log_data[62].valid := 1, [31].log_data[63].valid := 1, [31].log_data[64].valid := 1, [31].log_data[65].valid := 1, [31].log_data[66].valid := 1, [31].log_data[67].valid := 1, [31].log_data[68].valid := 1, [31].log_data[69].valid := 1, [31].log_data[70].valid := 1, [31].log_data[71].valid := 1, [31].log_data[72].valid := 1, [31].log_data[73].valid := 1, [31].log_data[74].valid := 1, [31].log_data[75].valid := 1, [31].log_data[76].valid := 1, [31].log_data[77].valid := 1, [31].log_data[78].valid := 1, [31].log_data[79].valid := 1, [31].log_data[80].valid := 1, [31].log_data[81].valid := 1, [31].log_data[82].valid := 1, [31].log_data[83].valid := 1, [31].log_data[84].valid := 1, [31].log_data[85].valid := 1, [31].log_data[86].valid := 1, [31].log_data[87].valid := 1, [31].log_data[88].valid := 1, [31].log_data[89].valid := 1, [31].log_data[90].valid := 1, [31].log_data[91].valid := 1, [31].log_data[92].valid := 1, [31].log_data[93].valid := 1, [31].log_data[94].valid := 1, [31].log_data[95].valid := 1, [31].log_data[96].valid := 1, [31].log_data[97].valid := 1, [31].log_data[98].valid := 1, [31].log_data[99].valid := 1, [31].log_data[100].valid := 1, [31].log_data[101].valid := 1, [31].log_data[102].valid := 1, [31].log_data[103].valid := 1, [31].log_data[104].valid := 1, [31].log_data[105].valid := 1, [31].log_data[106].valid := 1, [31].log_data[107].valid := 1, [31].log_data[108].valid := 1, [31].log_data[109].valid := 1, [31].log_data[110].valid := 1, [31].log_data[111].valid := 1, [31].log_data[112].valid := 1, [31].log_data[113].valid := 1, [31].log_data[114].valid := 1, [31].log_data[115].valid := 1,
        [31].log_data[116].valid := 1, [31].log_data[117].valid := 1, [31].log_data[118].valid := 1, [31].log_data[119].valid := 1, [31].log_data[120].valid := 1, [31].log_data[121].valid := 1, [31].log_data[122].valid := 1, [31].log_data[123].valid := 1, [31].log_data[124].valid := 1, [31].time.Year := 2023, [31].time.Month := 1, [31].time.Day := 14, [31].time.Hour := 10, [31].time.Minute := 59, [31].time.Second := 59, [32].log_data[0].min := 1.0, [32].log_data[0].max := 1.0, [32].log_data[0].total := 3600.0, [32].log_data[0].time := 3600.0, [32].log_data[0].valid := 1, [32].log_data[1].max := 1.0, [32].log_data[1].total := 550.5, [32].log_data[1].time := 3600.0, [32].log_data[1].maxminute := 43, [32].log_data[1].valid := 1, [32].log_data[2].max := 1.0, [32].log_data[2].total := 547.0, [32].log_data[2].time := 3600.0, [32].log_data[2].maxminute := 43, [32].log_data[2].valid := 1, [32].log_data[3].time := 3600.0, [32].log_data[3].valid := 1, [32].log_data[4].time := 3600.0, [32].log_data[4].valid := 1, [32].log_data[5].max := 1.0, [32].log_data[5].total := 248.0, [32].log_data[5].time := 3600.0, [32].log_data[5].maxminute := 45, [32].log_data[5].valid := 1, [32].log_data[6].time := 3600.0, [32].log_data[6].valid := 1, [32].log_data[7].time := 3600.0, [32].log_data[7].valid := 1, [32].log_data[8].min := 1.0, [32].log_data[8].max := 1.0, [32].log_data[8].total := 3600.0, [32].log_data[8].time := 3600.0, [32].log_data[8].valid := 1, [32].log_data[9].min := 1.0, [32].log_data[9].max := 1.0, [32].log_data[9].total := 3600.0, [32].log_data[9].time := 3600.0, [32].log_data[9].valid := 1, [32].log_data[10].min := 1.0, [32].log_data[10].max := 1.0, [32].log_data[10].total := 3600.0, [32].log_data[10].time := 3600.0, [32].log_data[10].valid := 1, [32].log_data[11].time := 3600.0, [32].log_data[11].valid := 1,
        [32].log_data[12].min := 1.0, [32].log_data[12].max := 1.0, [32].log_data[12].total := 3600.0, [32].log_data[12].time := 3600.0, [32].log_data[12].valid := 1, [32].log_data[13].min := 1.0, [32].log_data[13].max := 1.0, [32].log_data[13].total := 3600.0, [32].log_data[13].time := 3600.0, [32].log_data[13].valid := 1, [32].log_data[14].time := 3600.0, [32].log_data[14].valid := 1, [32].log_data[15].time := 3600.0, [32].log_data[15].valid := 1, [32].log_data[16].time := 3600.0, [32].log_data[16].valid := 1, [32].log_data[17].min := 1.0, [32].log_data[17].max := 1.0, [32].log_data[17].total := 3600.0, [32].log_data[17].time := 3600.0, [32].log_data[17].valid := 1, [32].log_data[18].time := 3600.0, [32].log_data[18].valid := 1, [32].log_data[19].time := 3600.0, [32].log_data[19].valid := 1, [32].log_data[20].time := 3600.0, [32].log_data[20].valid := 1, [32].log_data[21].min := 1.0, [32].log_data[21].max := 1.0, [32].log_data[21].total := 3600.0, [32].log_data[21].time := 3600.0, [32].log_data[21].valid := 1, [32].log_data[22].time := 3600.0, [32].log_data[22].valid := 1, [32].log_data[23].time := 3600.0, [32].log_data[23].valid := 1, [32].log_data[24].time := 3600.0, [32].log_data[24].valid := 1, [32].log_data[25].time := 3600.0, [32].log_data[25].valid := 1, [32].log_data[26].time := 3600.0, [32].log_data[26].valid := 1, [32].log_data[27].time := 3600.0, [32].log_data[27].valid := 1, [32].log_data[28].time := 3600.0, [32].log_data[28].valid := 1, [32].log_data[29].min := 1.0, [32].log_data[29].max := 1.0, [32].log_data[29].total := 3600.0, [32].log_data[29].time := 3600.0, [32].log_data[29].valid := 1, [32].log_data[30].min := 1.0, [32].log_data[30].max := 1.0, [32].log_data[30].total := 3600.0, [32].log_data[30].time := 3600.0, [32].log_data[30].valid := 1, [32].log_data[31].max := 1.0, [32].log_data[31].total := 1474.2471, [32].log_data[31].time := 3600.0, [32].log_data[31].maxminute := 11,
        [32].log_data[31].valid := 1, [32].log_data[32].max := 1.0, [32].log_data[32].total := 1629.7471, [32].log_data[32].time := 3600.0, [32].log_data[32].valid := 1, [32].log_data[33].time := 3600.0, [32].log_data[33].valid := 1, [32].log_data[34].time := 3600.0, [32].log_data[34].valid := 1, [32].log_data[35].max := 1.0, [32].log_data[35].total := 1629.7471, [32].log_data[35].time := 3600.0, [32].log_data[35].maxminute := 5, [32].log_data[35].valid := 1, [32].log_data[36].max := 1.0, [32].log_data[36].total := 1440.7471, [32].log_data[36].time := 3600.0, [32].log_data[36].minminute := 4, [32].log_data[36].valid := 1, [32].log_data[37].max := 7.6384163, [32].log_data[37].total := 3647.975, [32].log_data[37].time := 3600.0, [32].log_data[37].maxminute := 45, [32].log_data[37].valid := 1, [32].log_data[38].time := 3600.0, [32].log_data[38].valid := 1, [32].log_data[39].min := 0.9982394, [32].log_data[39].max := 1.0210879, [32].log_data[39].total := 3632.29, [32].log_data[39].time := 3600.0, [32].log_data[39].minminute := 47, [32].log_data[39].maxminute := 49, [32].log_data[39].valid := 1, [32].log_data[40].min := 7.5544233, [32].log_data[40].max := 7.604438, [32].log_data[40].total := 27289.459, [32].log_data[40].time := 3600.0, [32].log_data[40].minminute := 58, [32].log_data[40].maxminute := 28, [32].log_data[40].valid := 1, [32].log_data[41].min := 0.030784423, [32].log_data[41].max := 0.045309816, [32].log_data[41].total := 137.49794, [32].log_data[41].time := 3600.0, [32].log_data[41].minminute := 28, [32].log_data[41].valid := 1, [32].log_data[42].min := 2.2923493, [32].log_data[42].max := 2.297178, [32].log_data[42].total := 8262.189, [32].log_data[42].time := 3600.0, [32].log_data[42].minminute := 51, [32].log_data[42].maxminute := 1, [32].log_data[42].valid := 1, [32].log_data[43].min := -0.26000214, [32].log_data[43].max := -0.26000214, [32].log_data[43].total := -935.9732, [32].log_data[43].time := 3600.0, [32].log_data[43].valid := 1, [32].log_data[44].min := -0.30000305, [32].log_data[44].max := -0.27999878,
